# B&R Automation Studio project KeePakST401VersionX (part 4)

#### MbApp.st - Implementation code
```iecst
(********************************************************************
 * COPYRIGHT -- Bernecker + Rainer
 ********************************************************************
 * Program: MbApp
 * File: MbApp.st
 * Author: Bernecker + Rainer
 * Created: October 22, 2009
 ********************************************************************
 * Implementation of program MbApp
 * State Nomenclature: "request" is a write to the nordson melter asking for some data
 * 					   "read" is a read from the nordson melter of the previously requested data
 *                     "write" is a write to the nordson melter asking to write some data to the melter
 *                     "verify" is a read from the nordson melter where we check to see that the write was accepted
 ********************************************************************)

PROGRAM _INIT

	NordsonTxPacket.Byte0_MelterControl := 16#1;
	NordsonTxPacket.Byte1_Command := 3;
	NordsonTxPacket.Byte2_Data_Index := 16#78;
	NordsonTxPacket.Byte3_Channel_Num := 16#3;
	NordsonTxPacket.Byte4_5_WriteData := 0;
	NordsonTxPacket.Byte6_7_Mot1Spd := 0;
	NordsonTxPacket.Byte8_9_Mot2Spd := 0;
	NordsonTxPacket.Byte10_11_Mot3Spd := 0;
	NordsonTxPacket.Byte12_13_Mot4Spd := 0;
	NordsonTxPacket.Byte14_15_NotUsed := 0;

	state := MB_IDLE;

	(* init values *)
	mb_station 			:= 'IF2.ST2';					(* path to modbus station *)
	write_register_address	:= 1024;						(* register address on modbus station *)
	read_register_address	:= 0;						(* register address on modbus station *)
	num_registers_to_write := 8;
	num_registers_to_read := 8;

	testChannel := CHANNEL_ACT_TEMP_START;
	testIdx := IDX_ACT_TEMP;

	gAdhesiveCtrlInterface.Commands.MelterOn := TRUE;
	gAdhesiveCtrlInterface.Commands.PumpsOn := TRUE;
	gAdhesiveCtrlInterface.Parameters.NordsonComms.StandbyTimeoutTime := T#2h;

	FirstTimeCopySetTemps := FALSE;

END_PROGRAM

PROGRAM _CYCLIC

	IF(gAdhesiveCtrlInterface.Parameters.FeedbackIsModbusTCP) THEN
		gHMI.StatusDatapoints.NordsonModbusSDP := UNHIDE + UNLOCK;
	ELSE
		gHMI.StatusDatapoints.NordsonModbusSDP := HIDE + LOCK;
	END_IF

	StandbyTimer.IN := NOT(gRamCtrlInterface.Status.Running) AND NOT(gAdhesiveCtrlInterface.Commands.MelterStandbyOn);
	StandbyTimer.PT := gAdhesiveCtrlInterface.Parameters.NordsonComms.StandbyTimeoutTime;
	StandbyTimer();

	IF(StandbyTimer.Q) THEN
		gAdhesiveCtrlInterface.Commands.MelterStandbyOn := TRUE;
	END_IF

	//clearing standby on command shiuld turn standby off. Changed standbyoff to True
	IF(gAdhesiveCtrlInterface.Commands.MelterStandbyOff) THEN
		gAdhesiveCtrlInterface.Commands.MelterStandbyOff := TRUE;
		gAdhesiveCtrlInterface.Commands.MelterStandbyOn := FALSE;
	END_IF

	IF((gAdhesiveCtrlInterface.Status.NordsonInStandby) AND (gAdhesiveCtrlInterface.Parameters.FeedbackIsModbusTCP)) THEN
		gHMI.StatusDatapoints.NordsonStandbyOffSDP := UNHIDE + UNLOCK;
	ELSE
		gHMI.StatusDatapoints.NordsonStandbyOffSDP := HIDE + LOCK;
	END_IF

	//if nordson feedback is bypassed, the error count should reset to 0
	IF gAdhesiveCtrlInterface.Parameters.NordsonComms.ByPassFeedback THEN
		gAdhesiveCtrlInterface.Parameters.NordsonComms.ConsecutiveErrorCount := 0;
	END_IF

	CASE state OF

		MB_IDLE:
			FeedbackCycleTimer.IN := ((gAdhesiveCtrlInterface.Parameters.FeedbackIsModbusTCP) AND (gAdhesiveCtrlInterface.Parameters.NordsonComms.ByPassFeedback = FALSE));

			IF(gAdhesiveCtrlInterface.Parameters.FeedbackIsModbusTCP = FALSE) THEN
				gAdhesiveCtrlInterface.Parameters.NordsonComms.ConsecutiveErrorCount := 0;
			END_IF

			IF(gAdhesiveCtrlInterface.Commands.WriteChannelTemp) THEN
				gAdhesiveCtrlInterface.Commands.WriteChannelTemp := FALSE;
				TempChannelToWrite := 0;
				state := MB_WRITE_SET_TEMP;

			ELSIF(FeedbackCycleTimer.Q) THEN
				FeedbackCycleTimer.IN := FALSE;
				state := MB_REQUEST_MELTER_STATUS;
			END_IF

		MB_REQUEST_MELTER_STATUS:

			WriteMultipleRegisters.enable := 1;
			NordsonTxPacket.Byte0_MelterControl := MelterCmd;
			NordsonTxPacket.Byte1_Command := READ_COMMAND;
			NordsonTxPacket.Byte2_Data_Index := IDX_MELTER_STATUS;
			NordsonTxPacket.Byte3_Channel_Num := 0;

			IF((WriteMultipleRegisters.status = ERR_FUB_ENABLE_FALSE) OR (WriteMultipleRegisters.status = ERR_FUB_BUSY)) THEN
				//do nothing
			ELSIF(WriteMultipleRegisters.status = ERR_OK) THEN
				WriteMultipleRegisters.enable := 0;
				state := MB_READ_MELTER_STATUS;
			ELSE
				WriteMultipleRegisters.enable := 0;
				MBError := WriteMultipleRegisters.status;
				state := MB_ERROR;
			END_IF

		MB_READ_MELTER_STATUS:

			ReadMultipleRegisters.enable := 1;

			IF((ReadMultipleRegisters.status = ERR_FUB_ENABLE_FALSE) OR (ReadMultipleRegisters.status = ERR_FUB_BUSY)) THEN
				//do nothing
			ELSIF(ReadMultipleRegisters.status = ERR_OK) THEN

				ReadMultipleRegisters.enable := 0;

				IF(NordsonRxPacket.Byte2_Ack_Data_Index = NordsonTxPacket.Byte2_Data_Index) THEN

					gAdhesiveCtrlInterface.Parameters.NordsonComms.MelterStatus := NordsonRxPacket.Byte4_5_Read_Data_0;
					gAdhesiveCtrlInterface.Parameters.NordsonComms.MelterIsOn := (gAdhesiveCtrlInterface.Parameters.NordsonComms.MelterStatus <> 8); //melter status == 8 => melter is not on

					DecodeStatus;

					//the melter MUST see a 0 for its ON command before it sees a 1. Send a 0 if the unit is faulted OR we have previously told it to turn on. and it never came on
				//	IF((gAdhesiveCtrlInterface.Parameters.NordsonComms.UnitFaulted) OR ((gAdhesiveCtrlInterface.Parameters.NordsonComms.MelterIsOn = FALSE) AND (NordsonTxPacket.Byte0_MelterControl.0 = TRUE))) THEN
					IF((gAdhesiveCtrlInterface.Parameters.NordsonComms.MelterIsOn = FALSE) AND (NordsonTxPacket.Byte0_MelterControl.0 = TRUE)) THEN
						MelterCmd := MELTER_OFF + PUMPS_OFF; //melter off, pumps off
					ELSE

						MelterCmd := 0;
						IF(gAdhesiveCtrlInterface.Commands.MelterOn) THEN
							MelterCmd := MelterCmd + MELTER_ON;
						END_IF

						IF((gAdhesiveCtrlInterface.Commands.PumpsOn) AND (gAdhesiveCtrlInterface.Status.UnitReady)) THEN
							MelterCmd := MelterCmd + PUMPS_ON; //only turn the pump on if the melter is ready
						END_IF

						IF((gAdhesiveCtrlInterface.Commands.MelterStandbyOn = FALSE) OR ((gAdhesiveCtrlInterface.Status.NordsonInStandby = FALSE) AND NordsonTxPacket.Byte0_MelterControl.6 = TRUE)) THEN
							//do not standby on
						ELSIF (gAdhesiveCtrlInterface.Commands.MelterStandbyOn = TRUE) THEN
							MelterCmd := MelterCmd + STANDBY_ON; //only turn the pump on if the melter is ready
						END_IF
					END_IF

					state := MB_REQUEST_SET_TEMPS;
				ELSE
					//stay in this state and re-execute read
				END_IF

			ELSE
				ReadMultipleRegisters.enable := 0;
				MBError := ReadMultipleRegisters.status;
				state := MB_ERROR;
			END_IF

		MB_REQUEST_SET_TEMPS:

			WriteMultipleRegisters.enable := 1;
			NordsonTxPacket.Byte0_MelterControl := MelterCmd;
			NordsonTxPacket.Byte1_Command := READ_COMMAND;
			NordsonTxPacket.Byte2_Data_Index := IDX_SET_TEMP;
			NordsonTxPacket.Byte3_Channel_Num := CHANNEL_SET_TEMP_START;

			IF((WriteMultipleRegisters.status = ERR_FUB_ENABLE_FALSE) OR (WriteMultipleRegisters.status = ERR_FUB_BUSY)) THEN
				//do nothing
			ELSIF(WriteMultipleRegisters.status = ERR_OK) THEN
				WriteMultipleRegisters.enable := 0;
				gAdhesiveCtrlInterface.Parameters.NordsonComms.ConsecutiveErrorCount := 0;
				state := MB_READ_SET_TEMPS;
			ELSE
				WriteMultipleRegisters.enable := 0;
				MBError := WriteMultipleRegisters.status;
				state := MB_ERROR;
			END_IF

		MB_READ_SET_TEMPS:

			ReadMultipleRegisters.enable := 1;

			IF((ReadMultipleRegisters.status = ERR_FUB_ENABLE_FALSE) OR (ReadMultipleRegisters.status = ERR_FUB_BUSY)) THEN
				//do nothing
			ELSIF(ReadMultipleRegisters.status = ERR_OK) THEN
				ReadMultipleRegisters.enable := 0;
				gAdhesiveCtrlInterface.Parameters.NordsonComms.ConsecutiveErrorCount := 0;

				IF((NordsonRxPacket.Byte2_Ack_Data_Index = NordsonTxPacket.Byte2_Data_Index) AND
					(NordsonRxPacket.Byte3_Ack_Channel_Num = NordsonTxPacket.Byte3_Channel_Num)) THEN

					DecodeStatus;

					gAdhesiveCtrlInterface.Parameters.NordsonComms.ChannelSetTempActual[0] := NordsonRxPacket.Byte4_5_Read_Data_0;
					gAdhesiveCtrlInterface.Parameters.NordsonComms.ChannelSetTempActual[1] := NordsonRxPacket.Byte6_7_Read_Data_1;
					gAdhesiveCtrlInterface.Parameters.NordsonComms.ChannelSetTempActual[2] := NordsonRxPacket.Byte8_9_Read_Data_2;
					gAdhesiveCtrlInterface.Parameters.NordsonComms.ChannelSetTempActual[3] := NordsonRxPacket.Byte10_11_Read_Data_3;
					gAdhesiveCtrlInterface.Parameters.NordsonComms.ChannelSetTempActual[4] := NordsonRxPacket.Byte12_13_Read_Data_4;
					gAdhesiveCtrlInterface.Parameters.NordsonComms.ChannelSetTempActual[5] := NordsonRxPacket.Byte14_15_Read_Data_5;

					IF (FirstTimeCopySetTemps = FALSE) THEN
						gAdhesiveCtrlInterface.Parameters.NordsonComms.ChannelSetTempRequested := gAdhesiveCtrlInterface.Parameters.NordsonComms.ChannelSetTempActual;
						FirstTimeCopySetTemps := TRUE;
					END_IF

					state := MB_REQUEST_ACT_TEMPS; //for now, just go back to idle. Future versions need to read more stuff
				ELSE
					//stay in this state and re-execute read
				END_IF
			ELSE
				ReadMultipleRegisters.enable := 0;
				MBError := ReadMultipleRegisters.status;
				state := MB_ERROR;
			END_IF

		MB_REQUEST_ACT_TEMPS:

			WriteMultipleRegisters.enable := 1;
			NordsonTxPacket.Byte0_MelterControl := MelterCmd;
			NordsonTxPacket.Byte1_Command := READ_COMMAND;
			NordsonTxPacket.Byte2_Data_Index := IDX_ACT_TEMP;
			NordsonTxPacket.Byte3_Channel_Num := CHANNEL_ACT_TEMP_START;

			IF((WriteMultipleRegisters.status = ERR_FUB_ENABLE_FALSE) OR (WriteMultipleRegisters.status = ERR_FUB_BUSY)) THEN
				//do nothing
			ELSIF(WriteMultipleRegisters.status = ERR_OK) THEN
				WriteMultipleRegisters.enable := 0;
				state := MB_READ_ACT_TEMPS;
			ELSE
				WriteMultipleRegisters.enable := 0;
				MBError := WriteMultipleRegisters.status;
				state := MB_ERROR;
			END_IF

		MB_READ_ACT_TEMPS:

			ReadMultipleRegisters.enable := 1;

			IF((ReadMultipleRegisters.status = ERR_FUB_ENABLE_FALSE) OR (ReadMultipleRegisters.status = ERR_FUB_BUSY)) THEN
				//do nothing
			ELSIF(ReadMultipleRegisters.status = ERR_OK) THEN
				ReadMultipleRegisters.enable := 0;

				IF((NordsonRxPacket.Byte2_Ack_Data_Index = NordsonTxPacket.Byte2_Data_Index) AND
					(NordsonRxPacket.Byte3_Ack_Channel_Num = NordsonTxPacket.Byte3_Channel_Num)) THEN

					DecodeStatus;

					gAdhesiveCtrlInterface.Parameters.NordsonComms.ChannelActTemp[0] := NordsonRxPacket.Byte4_5_Read_Data_0;
					gAdhesiveCtrlInterface.Parameters.NordsonComms.ChannelActTemp[1] := NordsonRxPacket.Byte6_7_Read_Data_1;
					gAdhesiveCtrlInterface.Parameters.NordsonComms.ChannelActTemp[2] := NordsonRxPacket.Byte8_9_Read_Data_2;
					gAdhesiveCtrlInterface.Parameters.NordsonComms.ChannelActTemp[3] := NordsonRxPacket.Byte10_11_Read_Data_3;
					gAdhesiveCtrlInterface.Parameters.NordsonComms.ChannelActTemp[4] := NordsonRxPacket.Byte12_13_Read_Data_4;
					gAdhesiveCtrlInterface.Parameters.NordsonComms.ChannelActTemp[5] := NordsonRxPacket.Byte14_15_Read_Data_5;

					state := MB_REQUEST_ATS_ALARMS;
				ELSE
					//stay in this state and re-execute read
				END_IF

			ELSE
				ReadMultipleRegisters.enable := 0;
				MBError := ReadMultipleRegisters.status;
				state := MB_ERROR;
			END_IF

		MB_REQUEST_ATS_ALARMS:

			WriteMultipleRegisters.enable := 1;
			NordsonTxPacket.Byte0_MelterControl := MelterCmd;
			NordsonTxPacket.Byte1_Command := READ_COMMAND;
			NordsonTxPacket.Byte2_Data_Index := IDX_ATS_ALARMS;

			IF((WriteMultipleRegisters.status = ERR_FUB_ENABLE_FALSE) OR (WriteMultipleRegisters.status = ERR_FUB_BUSY)) THEN
				//do nothing
			ELSIF(WriteMultipleRegisters.status = ERR_OK) THEN
				WriteMultipleRegisters.enable := 0;
				state := MB_READ_ATS_ALARMS;
			ELSE
				WriteMultipleRegisters.enable := 0;
				MBError := WriteMultipleRegisters.status;
				state := MB_ERROR;
			END_IF

		MB_READ_ATS_ALARMS:

			ReadMultipleRegisters.enable := 1;

			IF((ReadMultipleRegisters.status = ERR_FUB_ENABLE_FALSE) OR (ReadMultipleRegisters.status = ERR_FUB_BUSY)) THEN
				//do nothing
			ELSIF(ReadMultipleRegisters.status = ERR_OK) THEN
				ReadMultipleRegisters.enable := 0;

				IF(NordsonRxPacket.Byte2_Ack_Data_Index = NordsonTxPacket.Byte2_Data_Index) THEN

					DecodeStatus;

					gAdhesiveCtrlInterface.Status.ATS_AddOnOverLimit := NordsonRxPacket.Byte4_5_Read_Data_0.0;
					gAdhesiveCtrlInterface.Status.ATS_AddOnUnderLimit := NordsonRxPacket.Byte4_5_Read_Data_0.1;

					state := MB_IDLE;
				ELSE
					//stay in this state and re-execute read
				END_IF

			ELSE
				ReadMultipleRegisters.enable := 0;
				MBError := ReadMultipleRegisters.status;
				state := MB_ERROR;
			END_IF

		MB_WRITE_SET_TEMP:

			WriteMultipleRegisters.enable := 1;
			NordsonTxPacket.Byte0_MelterControl := MelterCmd;
			NordsonTxPacket.Byte1_Command := WRITE_COMMAND;
			NordsonTxPacket.Byte2_Data_Index := IDX_SET_TEMP;
			NordsonTxPacket.Byte3_Channel_Num := TempChannelToWrite + 1; //TempChannelToWrite starts counting at 0, but nordson melter starts counting at 1
			NordsonTxPacket.Byte4_5_WriteData := gAdhesiveCtrlInterface.Parameters.NordsonComms.ChannelSetTempRequested[TempChannelToWrite];

			IF((WriteMultipleRegisters.status = ERR_FUB_ENABLE_FALSE) OR (WriteMultipleRegisters.status = ERR_FUB_BUSY)) THEN
				//do nothing
			ELSIF(WriteMultipleRegisters.status = ERR_OK) THEN
				WriteMultipleRegisters.enable := 0;
				state := MB_VERIFY_SET_TEMP_WRITE;
			ELSE
				WriteMultipleRegisters.enable := 0;
				MBError := WriteMultipleRegisters.status;
				state := MB_ERROR;
			END_IF

		MB_VERIFY_SET_TEMP_WRITE:

			ReadMultipleRegisters.enable := 1;

			IF((ReadMultipleRegisters.status = ERR_FUB_ENABLE_FALSE) OR (ReadMultipleRegisters.status = ERR_FUB_BUSY)) THEN
				//do nothing
			ELSIF(ReadMultipleRegisters.status = ERR_OK) THEN
				ReadMultipleRegisters.enable := 0;

				IF((NordsonRxPacket.Byte2_Ack_Data_Index = NordsonTxPacket.Byte2_Data_Index) AND
					(NordsonRxPacket.Byte3_Ack_Channel_Num = NordsonTxPacket.Byte3_Channel_Num)) THEN

					DecodeStatus;

					IF(TempChannelToWrite < NUM_NORDSON_TEMP_ZONES_M1) THEN
						IF(TempChannelToWrite = 0) THEN
							TempChannelToWrite := 2; //channel 0 and 1 get the same temp, no need to re-write channel 1
							state := MB_WRITE_SET_TEMP;
						ELSE
							TempChannelToWrite := TempChannelToWrite + 1; //set the temperature for the next channel (Skip channel 2). Machine has 3 total channels
							state := MB_WRITE_SET_TEMP;
						END_IF
					ELSE
						state := MB_IDLE;
					END_IF
				ELSE
					//stay in this state and re-execute read
				END_IF

			ELSE
				ReadMultipleRegisters.enable := 0;
				MBError := ReadMultipleRegisters.status;
				state := MB_ERROR;
			END_IF

		MB_REQUEST_ADH_USE:

			WriteMultipleRegisters.enable := 1;
			NordsonTxPacket.Byte0_MelterControl := MelterCmd;
			NordsonTxPacket.Byte1_Command := READ_COMMAND;
			NordsonTxPacket.Byte2_Data_Index := IDX_ADHESIVE_HOUR;
			NordsonTxPacket.Byte3_Channel_Num := CHANNEL_ADHESIVE_HOUR;

			IF((WriteMultipleRegisters.status = ERR_FUB_ENABLE_FALSE) OR (WriteMultipleRegisters.status = ERR_FUB_BUSY)) THEN
				//do nothing
			ELSIF(WriteMultipleRegisters.status = ERR_OK) THEN
				WriteMultipleRegisters.enable := 0;
				state := MB_READ_ACT_TEMPS;
			ELSE
				WriteMultipleRegisters.enable := 0;
				MBError := WriteMultipleRegisters.status;
				state := MB_ERROR;
			END_IF

		MB_READ_ADH_USE:

			ReadMultipleRegisters.enable := 1;

			IF((ReadMultipleRegisters.status = ERR_FUB_ENABLE_FALSE) OR (ReadMultipleRegisters.status = ERR_FUB_BUSY)) THEN
				//do nothing
			ELSIF(ReadMultipleRegisters.status = ERR_OK) THEN
				ReadMultipleRegisters.enable := 0;

				IF((NordsonRxPacket.Byte2_Ack_Data_Index = NordsonTxPacket.Byte2_Data_Index) AND
					(NordsonRxPacket.Byte3_Ack_Channel_Num = NordsonTxPacket.Byte3_Channel_Num)) THEN

					//	NordsonData.AdhesiveUsePerHour := NordsonRxPacket.Byte4_5_Read_Data_0 + (NordsonRxPacket.Byte6_7_Read_Data_1*(65536)); //data 0 + data 1 shifted up 16 bits

					state := MB_READ_ACT_TEMPS;
				ELSE
					//stay in this state and re-execute read
				END_IF
			END_IF

		MB_WRITE_REGISTERS:

			WriteMultipleRegisters.enable := 1;
			NordsonTxPacket.Byte0_MelterControl := MELTER_ON;
			NordsonTxPacket.Byte1_Command := READ_COMMAND;
			NordsonTxPacket.Byte2_Data_Index := testChannel;
			NordsonTxPacket.Byte3_Channel_Num := testIdx;

			IF((WriteMultipleRegisters.status = ERR_FUB_ENABLE_FALSE) OR (WriteMultipleRegisters.status = ERR_FUB_BUSY)) THEN
				//do nothing
			ELSIF(WriteMultipleRegisters.status = ERR_OK) THEN
				WriteMultipleRegisters.enable := 0;
				state := MB_READ_ACT_TEMPS;
			ELSE
				WriteMultipleRegisters.enable := 0;
				MBError := WriteMultipleRegisters.status;
				state := MB_ERROR;
			END_IF

		MB_READ_REGISTERS:

			ReadMultipleRegisters.enable := 1;

			IF((ReadMultipleRegisters.status = ERR_FUB_ENABLE_FALSE) OR (ReadMultipleRegisters.status = ERR_FUB_BUSY)) THEN
				//do nothing
			ELSIF(ReadMultipleRegisters.status = ERR_OK) THEN
				ReadMultipleRegisters.enable := 0;
				state := MB_IDLE;
			ELSE
				ReadMultipleRegisters.enable := 0;
				MBError := ReadMultipleRegisters.status;
				state := MB_ERROR;
			END_IF

		MB_ERROR:
			gAdhesiveCtrlInterface.Parameters.NordsonComms.ConsecutiveErrorCount := gAdhesiveCtrlInterface.Parameters.NordsonComms.ConsecutiveErrorCount + 1;
		state := MB_IDLE; //keep re-trying indefinetly, logic below will set/reset alarms alarm

	END_CASE;

	IF EDGEPOS(gAdhesiveCtrlInterface.Parameters.NordsonComms.ConsecutiveErrorCount >= 10) THEN
		MpAlarmXSet(gAlarmXCore, ALARM_NORDSON_COMMS);
	ELSIF EDGENEG(gAdhesiveCtrlInterface.Parameters.NordsonComms.ConsecutiveErrorCount >= 10)THEN
		MpAlarmXReset(gAlarmXCore, ALARM_NORDSON_COMMS);
	END_IF

	IF EDGEPOS(gAdhesiveCtrlInterface.Status.ATS_AddOnOverLimit) THEN
		MpAlarmXSet(gAlarmXCore, ALARM_ATS_OVERLIMIT);
	ELSIF EDGENEG(gAdhesiveCtrlInterface.Status.ATS_AddOnOverLimit)THEN
		MpAlarmXReset(gAlarmXCore, ALARM_ATS_OVERLIMIT);
	END_IF

	IF EDGEPOS(gAdhesiveCtrlInterface.Status.ATS_AddOnUnderLimit) THEN
		MpAlarmXSet(gAlarmXCore, ALARM_ATS_UNDERLIMIT);
	ELSIF EDGENEG(gAdhesiveCtrlInterface.Status.ATS_AddOnUnderLimit)THEN
		MpAlarmXReset(gAlarmXCore, ALARM_ATS_UNDERLIMIT);
	END_IF

	IF EDGEPOS(gAdhesiveCtrlInterface.Status.NordsonInStandby) THEN
		MpAlarmXSet(gAlarmXCore, ALARM_NORDSON_STANDBY);
	ELSIF EDGENEG(gAdhesiveCtrlInterface.Status.NordsonInStandby)THEN
		MpAlarmXReset(gAlarmXCore, ALARM_NORDSON_STANDBY);
	END_IF

	//force unit ready and unit faulted status flags if ModbusTCP control is selected and bypass is enabled
	IF(gAdhesiveCtrlInterface.Parameters.FeedbackIsModbusTCP AND gAdhesiveCtrlInterface.Parameters.NordsonComms.ByPassFeedback) THEN
		gAdhesiveCtrlInterface.Parameters.NordsonComms.UnitReady := TRUE;
		gAdhesiveCtrlInterface.Parameters.NordsonComms.UnitFaulted := FALSE;
		gAdhesiveCtrlInterface.Status.ATS_AddOnOverLimit := FALSE;
		gAdhesiveCtrlInterface.Status.ATS_AddOnUnderLimit := FALSE;
	END_IF

	//Must be called after state machine. Do not move any function calls that are already below this line
	WriteMultipleRegisters.pStation := ADR(mb_station);
	WriteMultipleRegisters.startAddress := write_register_address;
	WriteMultipleRegisters.nrRegisters := num_registers_to_write;
	WriteMultipleRegisters.pData := ADR(NordsonTxPacket);
	WriteMultipleRegisters.dataSize := SIZEOF(NordsonTxPacket);
	WriteMultipleRegisters();

	ReadMultipleRegisters.pStation := ADR(mb_station);
	ReadMultipleRegisters.startAddress := read_register_address;
	ReadMultipleRegisters.nrRegisters := num_registers_to_read;
	ReadMultipleRegisters.pData := ADR(NordsonRxPacket);
	ReadMultipleRegisters.dataSize := SIZEOF(NordsonRxPacket);
	ReadMultipleRegisters();

	FeedbackCycleTimer.PT := gAdhesiveCtrlInterface.Parameters.NordsonComms.FeedbackTime;
	FeedbackCycleTimer();

				END_PROGRAM
```

#### MbApp.typ - Local data types
```iecst
(********************************************************************
 * COPYRIGHT -- Bernecker + Rainer
 ********************************************************************
 * Program: MbApp
 * File: MbApp.typ
 * Author: Bernecker + Rainer
 * Created: October 22, 2009
 ********************************************************************
 * Local data types of program MbApp
 ********************************************************************)

TYPE
	ModbusTCP_Handling_States_enum :
		(
		MB_IDLE := 0,
		MB_REQUEST_SET_TEMPS,
		MB_READ_SET_TEMPS,
		MB_REQUEST_ACT_TEMPS,
		MB_READ_ACT_TEMPS,
		MB_REQUEST_MELTER_STATUS,
		MB_READ_MELTER_STATUS,
		MB_REQUEST_ADH_USE,
		MB_READ_ADH_USE,
		MB_WRITE_REGISTERS,
		MB_READ_REGISTERS,
		MB_REQUEST_MACHINE_STATUS,
		MB_WRITE_SET_TEMP,
		MB_VERIFY_SET_TEMP_WRITE,
		MB_REQUEST_ATS_ALARMS,
		MB_READ_ATS_ALARMS,
		MB_ERROR := 999
		);
END_TYPE
```

#### MbApp.var - Local variables
```iecst
(********************************************************************
 * COPYRIGHT -- Bernecker + Rainer
 ********************************************************************
 * Program: MbApp
 * File: MbApp.var
 * Author: Bernecker + Rainer
 * Created: October 22, 2009
 ********************************************************************
 * Local variables of program MbApp
 ********************************************************************)
VAR
	state : ModbusTCP_Handling_States_enum;
	mb_station : STRING[50];
	write_register_address : UINT;
	num_registers_to_write : UINT;
	read_register_address : UINT;
	num_registers_to_read : UINT;
	ReadMultipleRegisters : mbReadHoldingRegisters;
	WriteMultipleRegisters : mbWriteMultipleRegisters;
	MBError : UINT;
	testIdx : USINT;
	NordsonRxPacket : NordsonRxPacket_typ;
	testChannel : USINT;
	NordsonTxPacket : NordsonTxPacket_typ;
	FeedbackCycleTimer : TON;
	MelterCmd : USINT;
	TempChannelToWrite : USINT;
	StandbyTimer : TON;
	FirstTimeCopySetTemps : BOOL;
END_VAR
```

#### Action.st
```iecst
ACTION DecodeStatus:

	gAdhesiveCtrlInterface.Parameters.NordsonComms.UnitReady := NordsonRxPacket.Byte0_1_Status.0; //status word description from nordson manual
	gAdhesiveCtrlInterface.Parameters.NordsonComms.PumpStartUpProtectionOn := NordsonRxPacket.Byte0_1_Status.1;
	gAdhesiveCtrlInterface.Parameters.NordsonComms.Alert := NordsonRxPacket.Byte0_1_Status.2;
	gAdhesiveCtrlInterface.Parameters.NordsonComms.UnitFaulted := NordsonRxPacket.Byte0_1_Status.3;
	gAdhesiveCtrlInterface.Parameters.NordsonComms.ShutDown := NordsonRxPacket.Byte0_1_Status.4;
	gAdhesiveCtrlInterface.Parameters.NordsonComms.HeatUpPhaseActive := NordsonRxPacket.Byte0_1_Status.5;
	gAdhesiveCtrlInterface.Status.NordsonInStandby := NordsonRxPacket.Byte0_1_Status.6;
	gAdhesiveCtrlInterface.Parameters.NordsonComms.CommFault := NordsonRxPacket.Byte0_1_Status.14;
	gAdhesiveCtrlInterface.Parameters.NordsonComms.CommFaultInDataValue := NordsonRxPacket.Byte0_1_Status.15;

END_ACTION
```

### Program Logical/Actuators/NordsonComm/NordsonExtendedComm (IEC)

#### MbPressure.st - Init, cyclic, exit code
```iecst
(*********************************************************************************
 * Copyright: B&R Industrial Automation GmbH
 * Author:    nealj
 * Created:   May 27, 2021/1:33 PM
 * This task will cyclicly read the current pressure and the tank level and will
 * write the pressure setpoints.
 *********************************************************************************)

PROGRAM _INIT

    Station              := 'IF2.ST2';
    ModbusRead.pStation  := ADR(Station);
    ModbusWrite.pStation := ADR(Station);

END_PROGRAM

PROGRAM _CYCLIC

    Channel.PressureSetpoint := PressureSetpoint;

    CASE ExtendedCommsState OF

        WORD_MANIPULATION:
            Channel.ActualPressure           := (UDINT_TO_REAL(Registers.ChannelActualPressureWord) / 1000);
            Tank.ActualLevel                    := Registers.TankActualLevelWord;
            Registers.ChannelSetPressureWord := REAL_TO_UDINT(Channel.PressureSetpoint * 1000);
            ExtendedCommsState                  := READ_ACTPRESS_W1;

        READ_ACTPRESS_W1:
            IF (ModbusRead.status = ERR_OK) THEN
                ModbusRead.enable  := FALSE;
                ExtendedCommsState := WRITE_SETPRESS_W1;
            ELSIF (ModbusRead.status = ERR_FUB_ENABLE_FALSE) THEN
                ModbusRead.startAddress := 6103;
                ModbusRead.nrRegisters  := 2;
                ModbusRead.pData        := ADR(Registers.ChannelActualPressureWord);
                ModbusRead.dataSize     := 8;
                ModbusRead.enable       := TRUE;
            END_IF

        WRITE_SETPRESS_W1:
            IF (ModbusWrite.status = ERR_OK) THEN
                ModbusWrite.enable  := FALSE;
                ExtendedCommsState := READ_TANKLEVEL_W1;
            ELSIF (ModbusRead.status = ERR_FUB_ENABLE_FALSE) AND (WriteFlag) THEN
                ModbusWrite.startAddress := 6203;
                ModbusWrite.nrRegisters  := 2;
                ModbusWrite.pData        := ADR(Registers.ChannelSetPressureWord);
                ModbusWrite.dataSize     := 8;
                ModbusWrite.enable       := TRUE;
                WriteFlag              := FALSE;
            ELSIF (ModbusWrite.status = ERR_FUB_ENABLE_FALSE) AND NOT(WriteFlag) THEN
                ExtendedCommsState := READ_TANKLEVEL_W1;
            END_IF

        READ_TANKLEVEL_W1:
            IF (ModbusRead.status = ERR_OK) THEN
                ModbusRead.enable := FALSE;
                ExtendedCommsState := WORD_MANIPULATION;
            ELSIF (ModbusWrite.status = ERR_FUB_ENABLE_FALSE) THEN
                ModbusRead.startAddress := 13002;
                ModbusRead.nrRegisters  := 1;
                ModbusRead.pData        := ADR(Registers.TankActualLevelWord);
                ModbusRead.dataSize     := 4;
                ModbusRead.enable       := TRUE;
            END_IF

        MODBUS_ERROR:
            IF ((ModbusRead.status = ERR_FUB_ENABLE_FALSE) AND (ModbusWrite.status = ERR_FUB_ENABLE_FALSE)) THEN
                ExtendedCommsState := WORD_MANIPULATION;
            ELSE
                ReadErrorNumber    := ModbusRead.status;
                WriteErrorNumber   := ModbusWrite.status;
                ModbusRead.enable  := FALSE;
                ModbusWrite.enable := FALSE;
            END_IF

    END_CASE

    IF ((ModbusRead.status > 0) AND (ModbusRead.status < 65534)) OR ((ModbusWrite.status > 0) AND (ModbusWrite.status < 65534)) THEN
        ExtendedCommsState := MODBUS_ERROR;
    END_IF

    //Call FUBs
    ModbusRead();
    ModbusWrite();

END_PROGRAM

PROGRAM _EXIT

END_PROGRAM
```

#### Types.typ - Local data types
```iecst
TYPE
	ExtendedComms_enum :
		(
		WORD_MANIPULATION,
		READ_ACTPRESS_W1,
		READ_ACTPRESS_W2,
		READ_ACTPRESS_W3,
		READ_ACTPRESS_W4,
		WRITE_SETPRESS_W1,
		WRITE_SETPRESS_W2,
		WRITE_SETPRESS_W3,
		WRITE_SETPRESS_W4,
		READ_TANKLEVEL_W1,
		MODBUS_ERROR
		);
END_TYPE
```

#### Variables.var - Local variables
```iecst
VAR
	ModbusRead : mbReadHoldingRegisters;
	ModbusWrite : mbWriteMultipleRegisters;
	Station : STRING[10];
	Registers : Register_typ;
	Channel : Channel_typ;
	PressureSetpoint : REAL;
	Tank : Tank_typ;
	ExtendedCommsState : ExtendedComms_enum;
	WriteFlag : BOOL;
	ReadErrorNumber : UINT;
	WriteErrorNumber : UINT;
	New_Variable : USINT;
END_VAR
```

### Program Logical/Actuators/FlexTest (IEC)

#### Variables.var
```iecst
VAR
	FB_NDSN_MB_PBFlex_Proc : FB_NDSN_MB_PBFlex_Process;
	FB_NDSN_MB_PBFlex_Ctrl : FB_NDSN_MB_PBFlex_CtrlSts;
	mb_Station : STRING[30];
END_VAR
```

#### Main.st
```iecst
PROGRAM _INIT
	(* Insert code here *)
	b_ModuleStatus;
	mb_Station 			:= 'IF2.ST2';
    Melter;
 //   FB_NDSN_MB_PBFlex_Ctrl;
 //   FB_NDSN_MB_PBFlex_Proc;
END_PROGRAM

PROGRAM _CYCLIC
	(* Insert code here *)
//	FB_NDSN_MB_PBFlex_Ctrl(IN_b_Enable :=NOT  Melter.b_r_LostCommunication,	IN_mb_station := mb_Station,Melter := Melter);
//  FB_NDSN_MB_PBFlex_Proc(IN_b_Enable :=NOT  Melter.b_r_LostCommunication, IN_mb_station := mb_Station,Melter := Melter);
//  Melter.b_r_LostCommunication :=NOT b_ModuleStatus;

    FB_NDSN_MB_PBFlex_Ctrl(IN_b_Enable := NOT Melter.b_r_LostCommunication , IN_mb_station := mb_Station , Melter := Melter );
    FB_NDSN_MB_PBFlex_Proc(IN_b_Enable := NOT Melter.b_r_LostCommunication , IN_mb_station := mb_Station , Melter := Melter );
    Melter.b_r_LostCommunication := NOT b_ModuleStatus;

END_PROGRAM

PROGRAM _EXIT
	(* Insert code here *)

END_PROGRAM
```

### Program Logical/Recipes/Recipes (IEC)

#### Variables.var
```iecst
VAR
	LastRecipeLoaded : STRING[80];
	MpRecipeXml_0 : MpRecipeXml;
	MpRecipeRegPar_0 : MpRecipeRegPar;
	MpRecipeRegPar_1 : MpRecipeRegPar;
	MpRecipeRegPar_2 : MpRecipeRegPar;
	MpRecipeRegPar_3 : MpRecipeRegPar;
	MpRecipeRegPar_4 : MpRecipeRegPar;
	MpRecipeRegPar_5 : MpRecipeRegPar;
	RegParActive0 : BOOL;
	RegParActive1 : BOOL;
	RegParActive2 : BOOL;
	RegParActive3 : BOOL;
	RegParActive4 : BOOL;
	RegParActive5 : BOOL;
	AllParsRegistered : BOOL;
END_VAR
```

#### Cyclic.ld
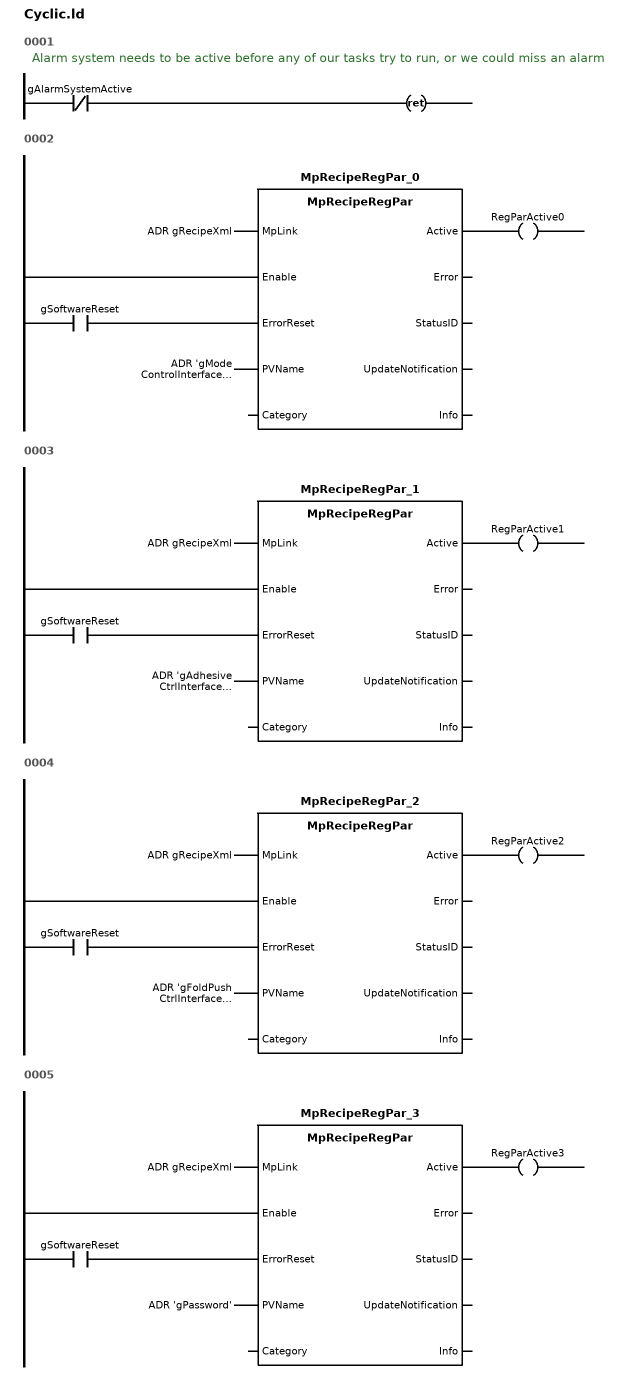
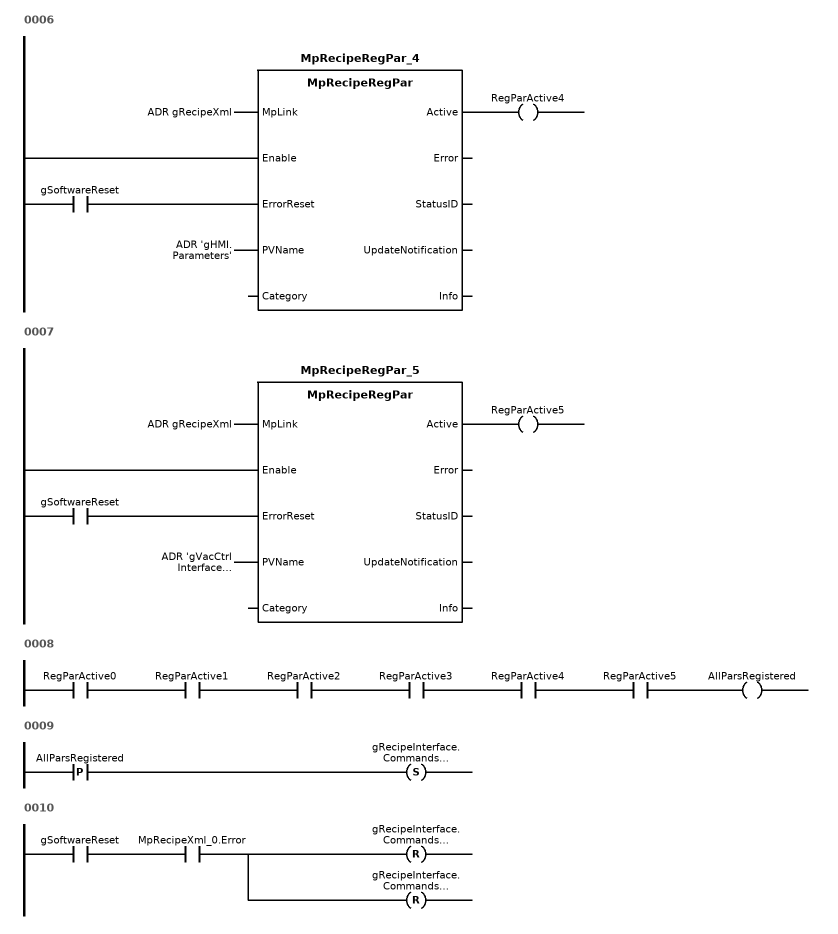
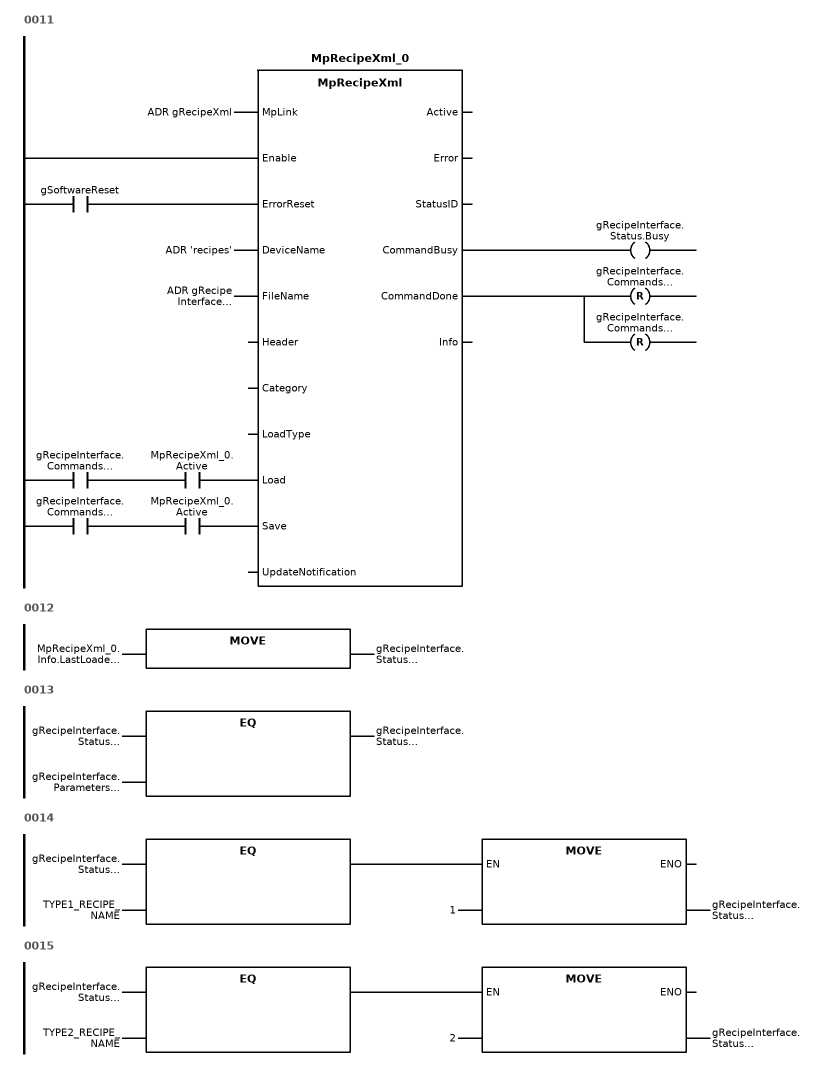
Ladder, written as Structured Text:
```iecst
PROGRAM _CYCLIC
VAR
    _e1 : R_TRIG;
    _p2 : BOOL;
    _p3 : BOOL;
END_VAR
(* Network 1: Alarm system needs to be active before any of our tasks try to run, or we could miss an alarm *)
IF NOT gAlarmSystemActive THEN RETURN; END_IF;

(* Network 2 *)
MpRecipeRegPar_0(MpLink := ADR(gRecipeXml), Enable := TRUE, ErrorReset := gSoftwareReset, PVName := ADR('gModeControlInterface.Parameters'));
RegParActive0 := MpRecipeRegPar_0.Active;

(* Network 3 *)
MpRecipeRegPar_1(MpLink := ADR(gRecipeXml), Enable := TRUE, ErrorReset := gSoftwareReset, PVName := ADR('gAdhesiveCtrlInterface.Parameters'));
RegParActive1 := MpRecipeRegPar_1.Active;

(* Network 4 *)
MpRecipeRegPar_2(MpLink := ADR(gRecipeXml), Enable := TRUE, ErrorReset := gSoftwareReset, PVName := ADR('gFoldPushCtrlInterface.Parameters'));
RegParActive2 := MpRecipeRegPar_2.Active;

(* Network 5 *)
MpRecipeRegPar_3(MpLink := ADR(gRecipeXml), Enable := TRUE, ErrorReset := gSoftwareReset, PVName := ADR('gPassword'));
RegParActive3 := MpRecipeRegPar_3.Active;

(* Network 6 *)
MpRecipeRegPar_4(MpLink := ADR(gRecipeXml), Enable := TRUE, ErrorReset := gSoftwareReset, PVName := ADR('gHMI.Parameters'));
RegParActive4 := MpRecipeRegPar_4.Active;

(* Network 7 *)
MpRecipeRegPar_5(MpLink := ADR(gRecipeXml), Enable := TRUE, ErrorReset := gSoftwareReset, PVName := ADR('gVacCtrlInterface.Parameters'));
RegParActive5 := MpRecipeRegPar_5.Active;

(* Network 8 *)
AllParsRegistered := RegParActive0 AND RegParActive1 AND RegParActive2 AND RegParActive3 AND RegParActive4 AND RegParActive5;

(* Network 9 *)
_e1(CLK := AllParsRegistered);
IF _e1.Q THEN gRecipeInterface.Commands.LoadRecipe := TRUE; END_IF;

(* Network 10 *)
IF gSoftwareReset AND MpRecipeXml_0.Error THEN
    gRecipeInterface.Commands.LoadRecipe := FALSE;
    gRecipeInterface.Commands.SaveRecipe := FALSE;
END_IF;

(* Network 11 *)
MpRecipeXml_0(MpLink := ADR(gRecipeXml), Enable := TRUE, ErrorReset := gSoftwareReset, DeviceName := ADR('recipes'), FileName := ADR(gRecipeInterface.Parameters.RecipeName), Load := gRecipeInterface.Commands.LoadRecipe AND MpRecipeXml_0.Active, Save := gRecipeInterface.Commands.SaveRecipe AND MpRecipeXml_0.Active);
gRecipeInterface.Status.Busy := MpRecipeXml_0.CommandBusy;
IF MpRecipeXml_0.CommandDone THEN
    gRecipeInterface.Commands.LoadRecipe := FALSE;
    gRecipeInterface.Commands.SaveRecipe := FALSE;
END_IF;

(* Network 12 *)
gRecipeInterface.Status.LoadedRecipeName := MpRecipeXml_0.Info.LastLoadedRecipe;

(* Network 13 *)
gRecipeInterface.Status.RecipeHasBeenLoaded := gRecipeInterface.Status.LoadedRecipeName = gRecipeInterface.Parameters.RecipeName;

(* Network 14 *)
_p2 := gRecipeInterface.Status.LoadedRecipeName = TYPE1_RECIPE_NAME;
IF _p2 THEN gRecipeInterface.Status.LoadedRecipeIndex := 1; END_IF;

(* Network 15 *)
_p3 := gRecipeInterface.Status.LoadedRecipeName = TYPE2_RECIPE_NAME;
IF _p3 THEN gRecipeInterface.Status.LoadedRecipeIndex := 2; END_IF;
END_PROGRAM
```

#### Init.st
```iecst
PROGRAM _INIT
	(* Insert code here *)

	gRecipeInterface.Commands.LoadRecipe := 1; //load settings on startup

	IF gRecipeInterface.Parameters.RecipeName = '' THEN
		gRecipeInterface.Parameters.RecipeName := TYPE1_RECIPE_NAME;
	END_IF

	//If the last recipe was type 2, set file name to that recipe. Otherwise default to recipe 1 file name
//	IF LastRecipeLoaded = TYPE2_RECIPE_NAME THEN
//		gRecipeInterface.Parameters.RecipeName := TYPE2_RECIPE_NAME;
//	ELSE
//		gRecipeInterface.Parameters.RecipeName := TYPE1_RECIPE_NAME;
//	END_IF

END_PROGRAM
```

### Program Logical/Recipes/GluePattCtrl (IEC)

#### Cyclic.st - Cyclic code
```iecst
PROGRAM _CYCLIC

	SaveButton_RTrig.CLK := gRecipeInterface.Commands.SaveRecipe;

	IF SaveButton_RTrig.Q THEN
		gAdhesiveCtrlInterface.Parameters.SavedPatterns[gAdhesiveCtrlInterface.Parameters.PatternSelection].AdhesivePatterns := gAdhesiveCtrlInterface.Parameters.AdhesivePatterns;
	END_IF

	IF gHMI.StatusDatapoints.AdhesivePatternConfirmedSDP.0 THEN
		gAdhesiveCtrlInterface.Parameters.AdhesivePatterns := gAdhesiveCtrlInterface.Parameters.SavedPatterns[gAdhesiveCtrlInterface.Parameters.PatternSelection].AdhesivePatterns;
		gHMI.StatusDatapoints.AdhesivePatternConfirmedSDP.0 := FALSE;
	END_IF

    SaveButton_RTrig();

END_PROGRAM
```

#### Variables.var - Local variables
```iecst
VAR
	SaveButton_RTrig : R_TRIG;
END_VAR
```

### Program Logical/AlarmControl/AlarmHandling (IEC)

#### Cyclic.ld - Cyclic code
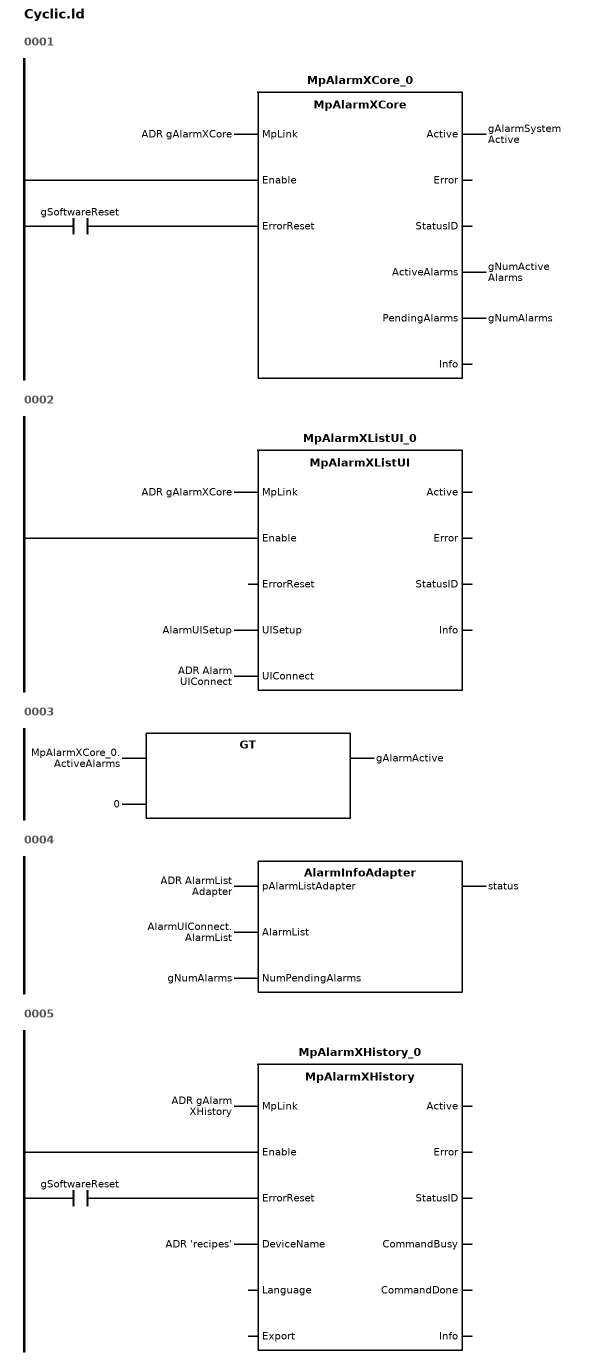
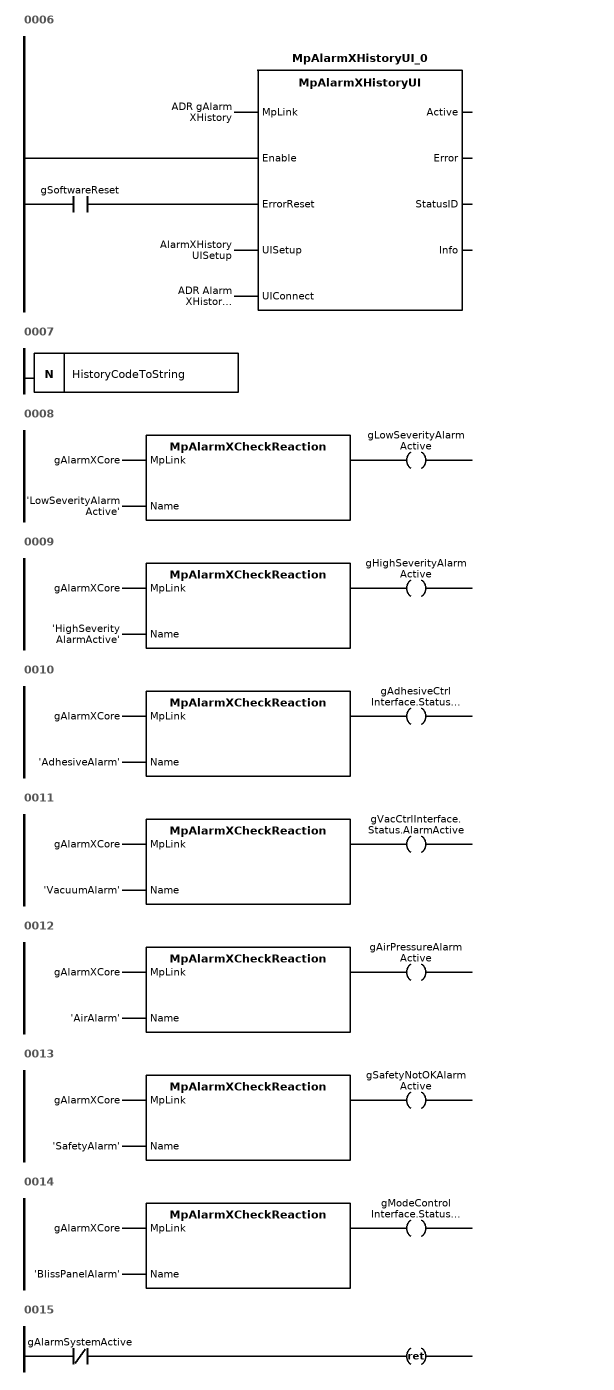
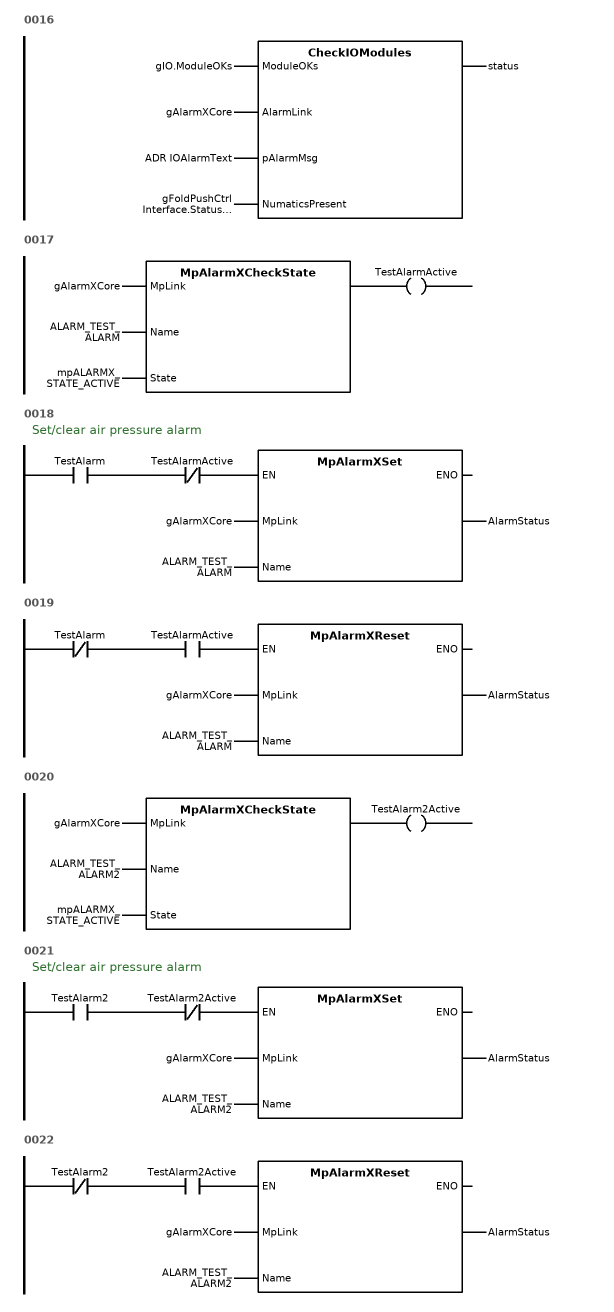
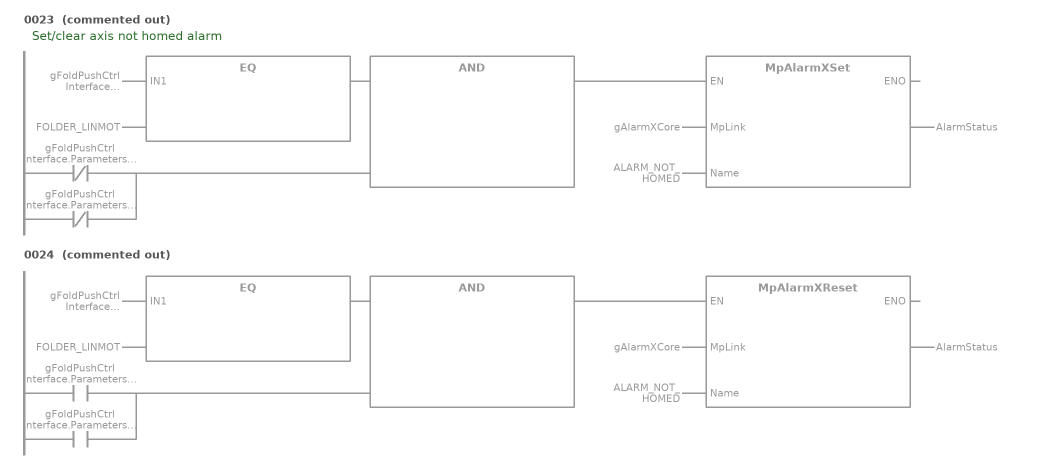
Ladder, written as Structured Text:
```iecst
PROGRAM _CYCLIC
(* Network 1 *)
MpAlarmXCore_0(MpLink := ADR(gAlarmXCore), Enable := TRUE, ErrorReset := gSoftwareReset);
gAlarmSystemActive := MpAlarmXCore_0.Active;
gNumActiveAlarms := MpAlarmXCore_0.ActiveAlarms;
gNumAlarms := MpAlarmXCore_0.PendingAlarms;

(* Network 2 *)
MpAlarmXListUI_0(MpLink := ADR(gAlarmXCore), Enable := TRUE, UISetup := AlarmUISetup, UIConnect := ADR(AlarmUIConnect));

(* Network 3 *)
gAlarmActive := MpAlarmXCore_0.ActiveAlarms > 0;

(* Network 4 *)
status := AlarmInfoAdapter(pAlarmListAdapter := ADR(AlarmListAdapter), AlarmList := AlarmUIConnect.AlarmList, NumPendingAlarms := gNumAlarms);

(* Network 5 *)
MpAlarmXHistory_0(MpLink := ADR(gAlarmXHistory), Enable := TRUE, ErrorReset := gSoftwareReset, DeviceName := ADR('recipes'));

(* Network 6 *)
MpAlarmXHistoryUI_0(MpLink := ADR(gAlarmXHistory), Enable := TRUE, ErrorReset := gSoftwareReset, UISetup := AlarmXHistoryUISetup, UIConnect := ADR(AlarmXHistoryUIConnect));

(* Network 7 *)
HistoryCodeToString;

(* Network 8 *)
gLowSeverityAlarmActive := MpAlarmXCheckReaction(MpLink := gAlarmXCore, Name := 'LowSeverityAlarmActive');

(* Network 9 *)
gHighSeverityAlarmActive := MpAlarmXCheckReaction(MpLink := gAlarmXCore, Name := 'HighSeverityAlarmActive');

(* Network 10 *)
gAdhesiveCtrlInterface.Status.AlarmActive := MpAlarmXCheckReaction(MpLink := gAlarmXCore, Name := 'AdhesiveAlarm');

(* Network 11 *)
gVacCtrlInterface.Status.AlarmActive := MpAlarmXCheckReaction(MpLink := gAlarmXCore, Name := 'VacuumAlarm');

(* Network 12 *)
gAirPressureAlarmActive := MpAlarmXCheckReaction(MpLink := gAlarmXCore, Name := 'AirAlarm');

(* Network 13 *)
gSafetyNotOKAlarmActive := MpAlarmXCheckReaction(MpLink := gAlarmXCore, Name := 'SafetyAlarm');

(* Network 14 *)
gModeControlInterface.Status.BlissPanelAlarmActive := MpAlarmXCheckReaction(MpLink := gAlarmXCore, Name := 'BlissPanelAlarm');

(* Network 15 *)
IF NOT gAlarmSystemActive THEN RETURN; END_IF;

(* Network 16 *)
status := CheckIOModules(ModuleOKs := gIO.ModuleOKs, AlarmLink := gAlarmXCore, pAlarmMsg := ADR(IOAlarmText), NumaticsPresent := gFoldPushCtrlInterface.Status.PowelinkConfig);

(* Network 17 *)
TestAlarmActive := MpAlarmXCheckState(MpLink := gAlarmXCore, Name := ALARM_TEST_ALARM, State := mpALARMX_STATE_ACTIVE);

(* Network 18: Set/clear air pressure alarm *)
IF TestAlarm AND NOT TestAlarmActive THEN
    AlarmStatus := MpAlarmXSet(MpLink := gAlarmXCore, Name := ALARM_TEST_ALARM);
END_IF;

(* Network 19 *)
IF NOT TestAlarm AND TestAlarmActive THEN
    AlarmStatus := MpAlarmXReset(MpLink := gAlarmXCore, Name := ALARM_TEST_ALARM);
END_IF;

(* Network 20 *)
TestAlarm2Active := MpAlarmXCheckState(MpLink := gAlarmXCore, Name := ALARM_TEST_ALARM2, State := mpALARMX_STATE_ACTIVE);

(* Network 21: Set/clear air pressure alarm *)
IF TestAlarm2 AND NOT TestAlarm2Active THEN
    AlarmStatus := MpAlarmXSet(MpLink := gAlarmXCore, Name := ALARM_TEST_ALARM2);
END_IF;

(* Network 22 *)
IF NOT TestAlarm2 AND TestAlarm2Active THEN
    AlarmStatus := MpAlarmXReset(MpLink := gAlarmXCore, Name := ALARM_TEST_ALARM2);
END_IF;

(* Network 23: Set/clear axis not homed alarm *) (* commented out *)
// IF (gFoldPushCtrlInterface.Parameters.FolderTypeSelection = FOLDER_LINMOT) AND (NOT gFoldPushCtrlInterface.Parameters.LinMotTopFolder.Status.IsHomed OR NOT gFoldPushCtrlInterface.Parameters.LinMotBotFolder.Status.IsHomed) THEN
//     AlarmStatus := MpAlarmXSet(MpLink := gAlarmXCore, Name := ALARM_NOT_HOMED);
// END_IF;

(* Network 24 *) (* commented out *)
// IF (gFoldPushCtrlInterface.Parameters.FolderTypeSelection = FOLDER_LINMOT) AND (gFoldPushCtrlInterface.Parameters.LinMotTopFolder.Status.IsHomed OR gFoldPushCtrlInterface.Parameters.LinMotBotFolder.Status.IsHomed) THEN
//     AlarmStatus := MpAlarmXReset(MpLink := gAlarmXCore, Name := ALARM_NOT_HOMED);
// END_IF;
END_PROGRAM
```

#### Init.st
```iecst
PROGRAM _INIT

	FOR i := 0 TO 99 DO
		gIO.ModuleOKs[i] := TRUE;
	END_FOR;

	IOAlarmText;

	AlarmXHistoryUISetup.AlarmListScrollWindow := 1;
	AlarmXHistoryUISetup.AlarmListSize := 6;

END_PROGRAM
```

#### Variables.var - Local variables
```iecst
VAR
	IOAlarmText : STRING[100];
	MpAlarmXCore_0 : MpAlarmXCore;
	MpAlarmXListUI_0 : MpAlarmXListUI;
	AlarmUISetup : MpAlarmXListUISetupType;
	AlarmUIConnect : MpAlarmXListUIConnectType;
	AlarmListAdapter : AlarmListAdapter_typ;
	AlarmHistoryListAdapter : AlarmListAdapter_typ;
	status : BOOL;
	i : UINT;
	MpAlarmXHistory_0 : MpAlarmXHistory;
	MpAlarmXHistoryUI_0 : MpAlarmXHistoryUI;
	AlarmXHistoryUIConnect : MpAlarmXHistoryUIConnectType;
	AlarmXHistoryUISetup : MpAlarmXHistoryUISetupType;
	AlarmStatus : DINT;
	TestAlarm2 : BOOL;
	TestAlarm : BOOL;
	TestAlarm2Active : BOOL;
	TestAlarmActive : BOOL;
END_VAR
```

#### LocalFunctions.fun
```iecst
FUNCTION AlarmInfoAdapter : BOOL (*Convert some alarm elements from Bool to Str*) (*$GROUP=User,$CAT=User,$GROUPICON=User.png,$CATICON=User.png*)
	VAR_INPUT
		pAlarmListAdapter : REFERENCE TO AlarmListAdapter_typ;
		AlarmList : MpAlarmXListUIAlarmListType;
		NumPendingAlarms : UDINT;
	END_VAR
	VAR
		i : UINT;
	END_VAR
END_FUNCTION

FUNCTION CheckIOModules : BOOL (*TODO: Add your comment here*) (*$GROUP=User,$CAT=User,$GROUPICON=User.png,$CATICON=User.png*)
	VAR_INPUT
		ModuleOKs : ARRAY[0..99] OF BOOL;
		AlarmLink : MpComIdentType;
		pAlarmMsg : UDINT;
	END_VAR
	VAR
		i : USINT;
	END_VAR
	VAR_INPUT
		NumaticsPresent : BOOL;
	END_VAR
END_FUNCTION
```

#### AlarmInfoAdapter.st
```iecst
(* Convert some alarm elements from Bool to Str *)
FUNCTION AlarmInfoAdapter

	IF(NumPendingAlarms = 0) THEN
		FOR i:= 0  TO 49 DO
			pAlarmListAdapter.Acknowledged[i] := '';
			pAlarmListAdapter.Active[i] := '';
			pAlarmListAdapter.Code[i] := '';
		END_FOR
	ELSE

		FOR i:=0 TO AlarmList.MaxSelection DO

			IF(AlarmList.StateAcknowledged[i] = TRUE) THEN
				pAlarmListAdapter.Acknowledged[i] := 'Yes';
			ELSE
				pAlarmListAdapter.Acknowledged[i] := 'No';
			END_IF

			IF(AlarmList.StateActive[i] = TRUE) THEN
				pAlarmListAdapter.Active[i] := 'Yes';
			ELSE
				pAlarmListAdapter.Active[i] := 'No';
			END_IF

			brsitoa(AlarmList.Code[i],ADR(pAlarmListAdapter.Code[i]));

		END_FOR;

		FOR i:= AlarmList.MaxSelection + 1  TO 49 DO
			pAlarmListAdapter.Acknowledged[i] := '';
			pAlarmListAdapter.Active[i] := '';
			pAlarmListAdapter.Code[i] := '';
		END_FOR

	END_IF

	AlarmInfoAdapter := TRUE;

END_FUNCTION
```

#### CheckIOModules.st
```iecst
(* TODO: Add your comment here *)
FUNCTION CheckIOModules

	brsmemset(pAlarmMsg, 0, 100);

	FOR i := 1 TO 99 DO

		IF(ModuleOKs[i] = FALSE) THEN

			IF (i = 1) THEN
				brsstrcat(pAlarmMsg, ADR ('Module 1 Bus Receiver'));
			ELSIF (i = 2) THEN
				brsstrcat(pAlarmMsg, ADR ('Module 2 DI 1'));
			ELSIF (i = 3) THEN
				brsstrcat(pAlarmMsg, ADR ('Module 3 D0 1'));
			ELSIF (i = 4) THEN
				brsstrcat(pAlarmMsg, ADR ('Module 4 DO 2(high wattage outputs)'));
			ELSIF (i = 5) THEN
				brsstrcat(pAlarmMsg, ADR ('Module 5 Encoder Inputs'));
			ELSIF (i = 6) THEN
				brsstrcat(pAlarmMsg, ADR ('SLX Module'));

			ELSIF (i = 7) THEN
				IF NumaticsPresent THEN
				brsstrcat(pAlarmMsg, ADR ('Module 7 Pneumatics 580'));
				END_IF

			END_IF

			IF (i=7 AND NumaticsPresent) OR (i<> 7) THEN
			brsstrcat(pAlarmMsg, ADR (' Not OK'));

			MpAlarmXSet(AlarmLink, ALARM_IO_MODULE_NOT_OK);
			END_IF

			RETURN;

		END_IF

	END_FOR;

	MpAlarmXReset(AlarmLink, ALARM_IO_MODULE_NOT_OK);

	CheckIOModules := 1;

END_FUNCTION
```

#### Action.st
```iecst
//convert alarm code integer into a string. This let's us completely clear alarm codes for empty entries instead of entering a '0'
ACTION HistoryCodeToString:

	FOR i:=0 TO AlarmXHistoryUIConnect.AlarmList.MaxSelection DO

		brsitoa(AlarmXHistoryUIConnect.AlarmList.Code[i], ADR(AlarmHistoryListAdapter.Code[i]));

	END_FOR;

	FOR i:= AlarmXHistoryUIConnect.AlarmList.MaxSelection + 1  TO 49 DO
		AlarmHistoryListAdapter.Code[i] := '';
	END_FOR

END_ACTION
```

### Program Logical/HMI/HMIControl (IEC)

#### Variables.var
```iecst
VAR
	FlashOFF : TON;
	FlashON : TON;
	status : BOOL;
	SettingsLoaded : BOOL;
	LogoutTimer : TON;
	OldPage : USINT;
	ResetTimeoutTimer : BOOL;
	ResetUserLevel : BOOL;
END_VAR
```

#### Cyclic.ld
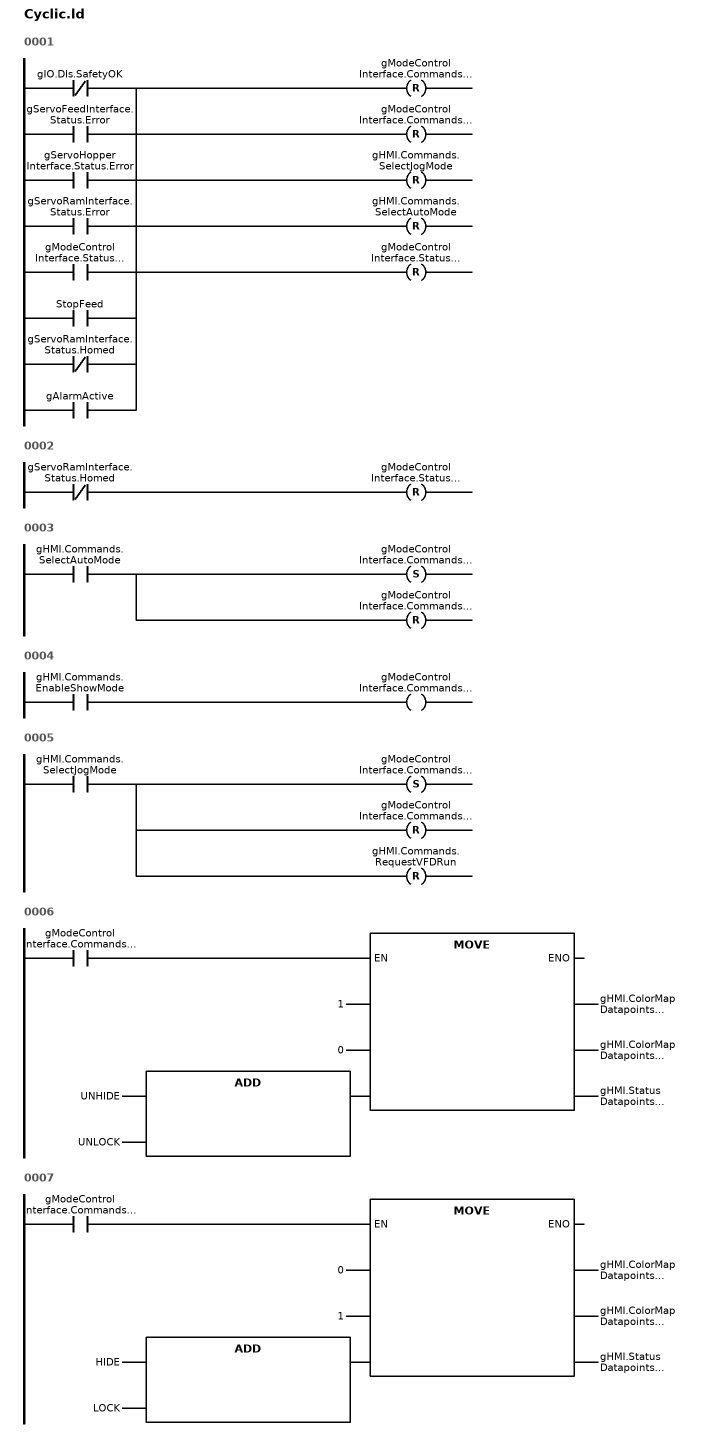
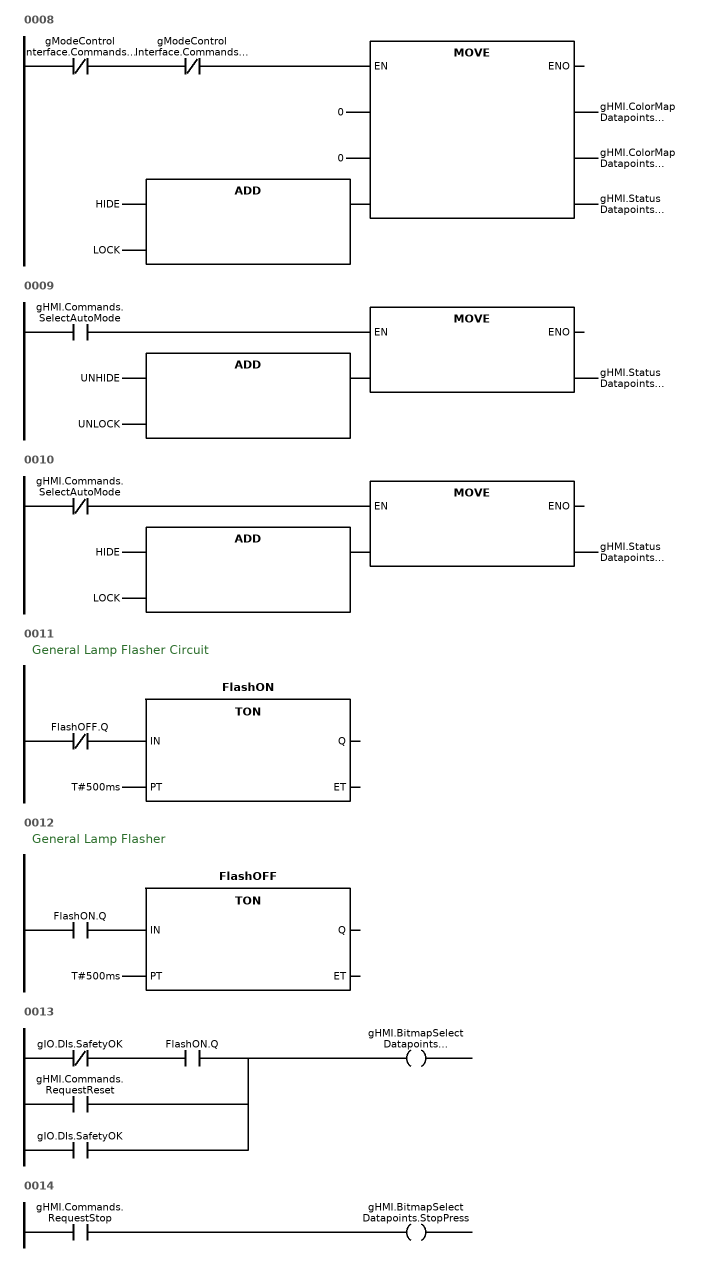
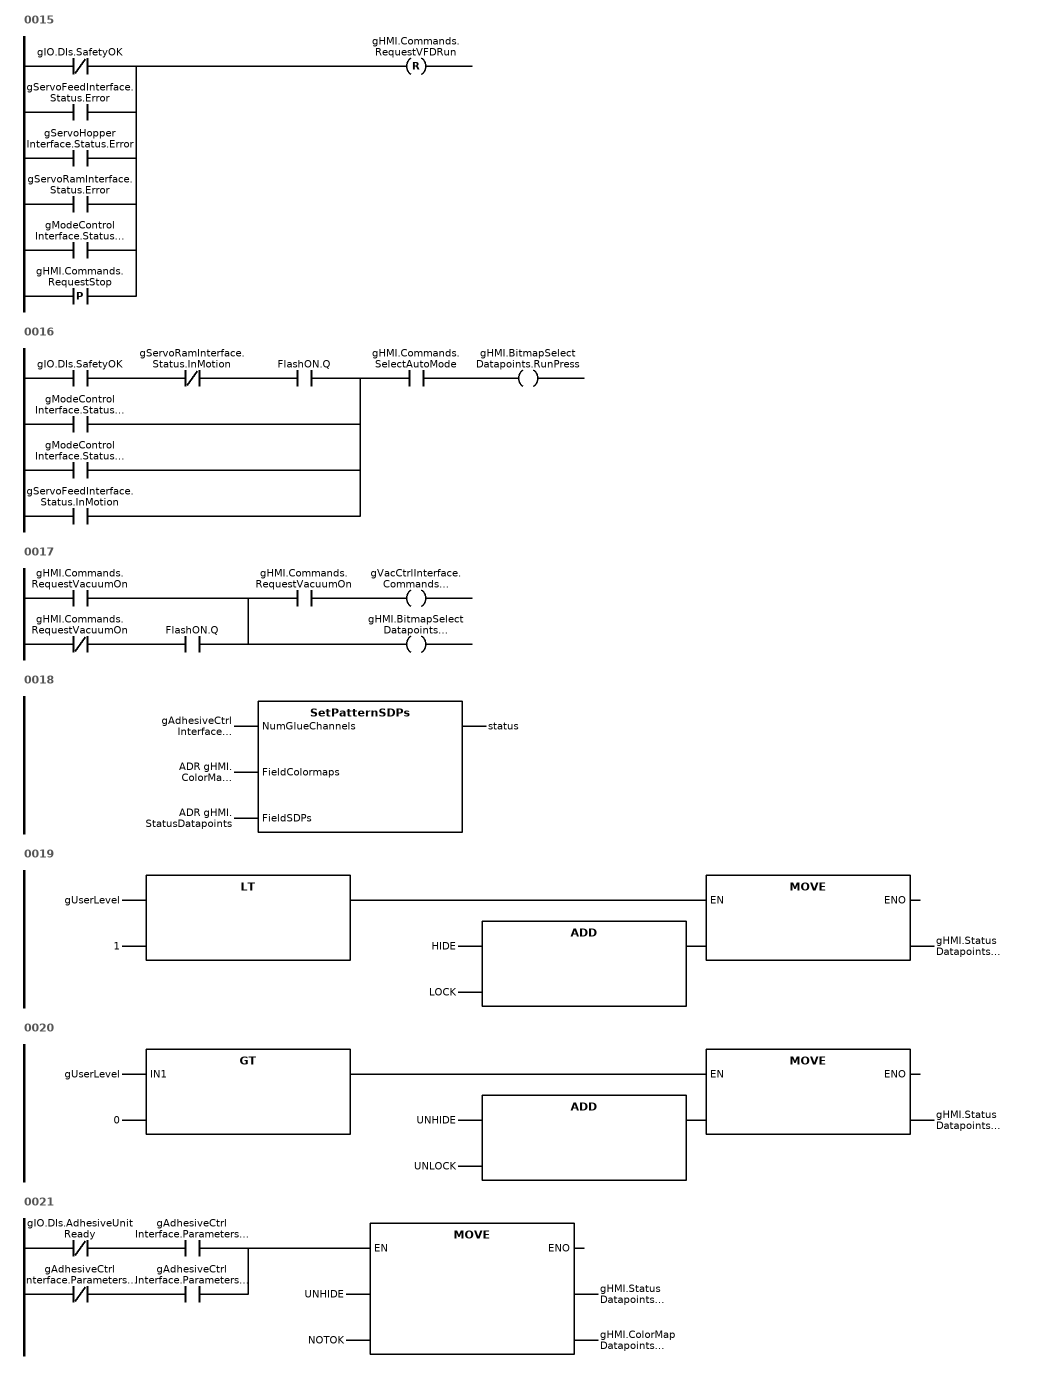
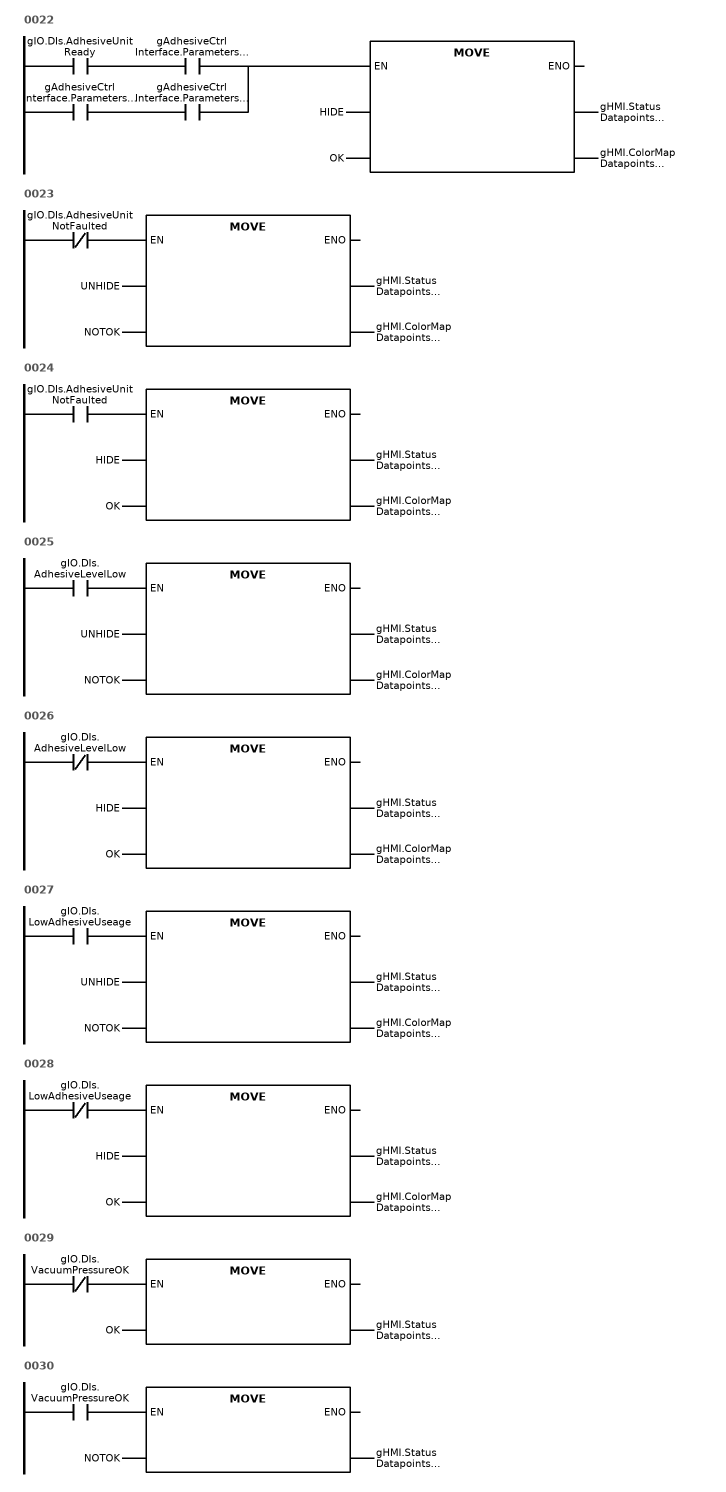
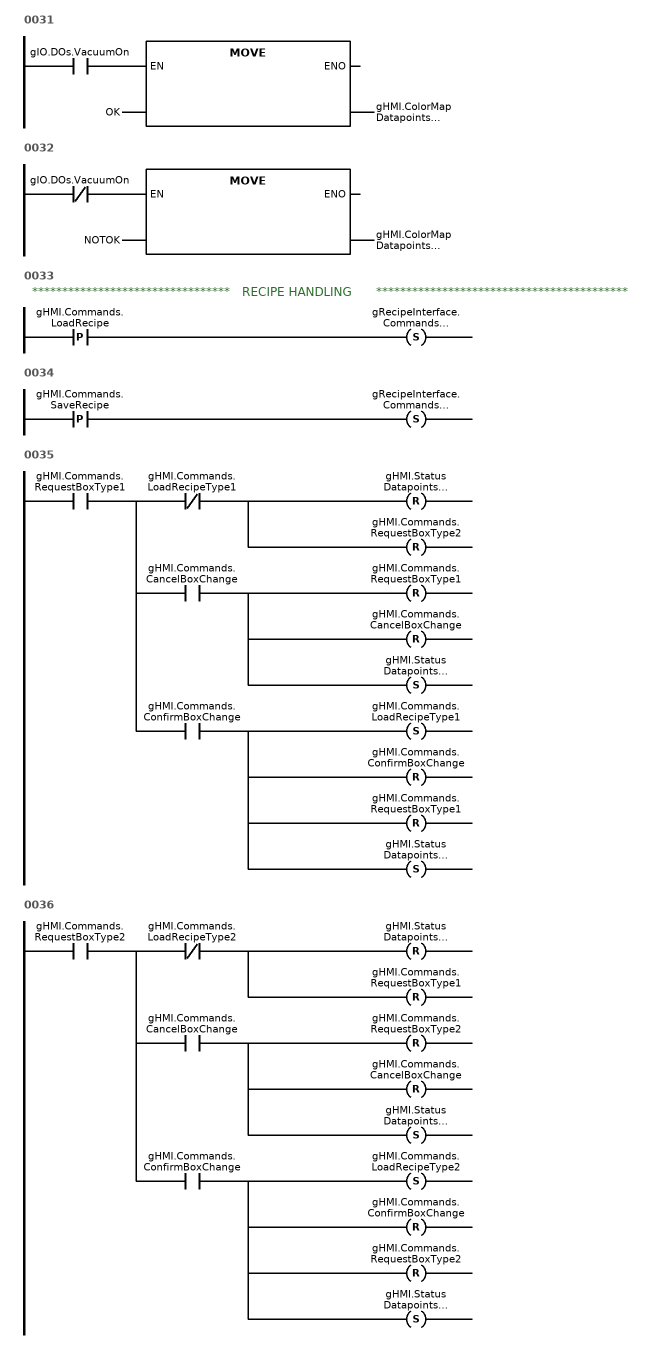
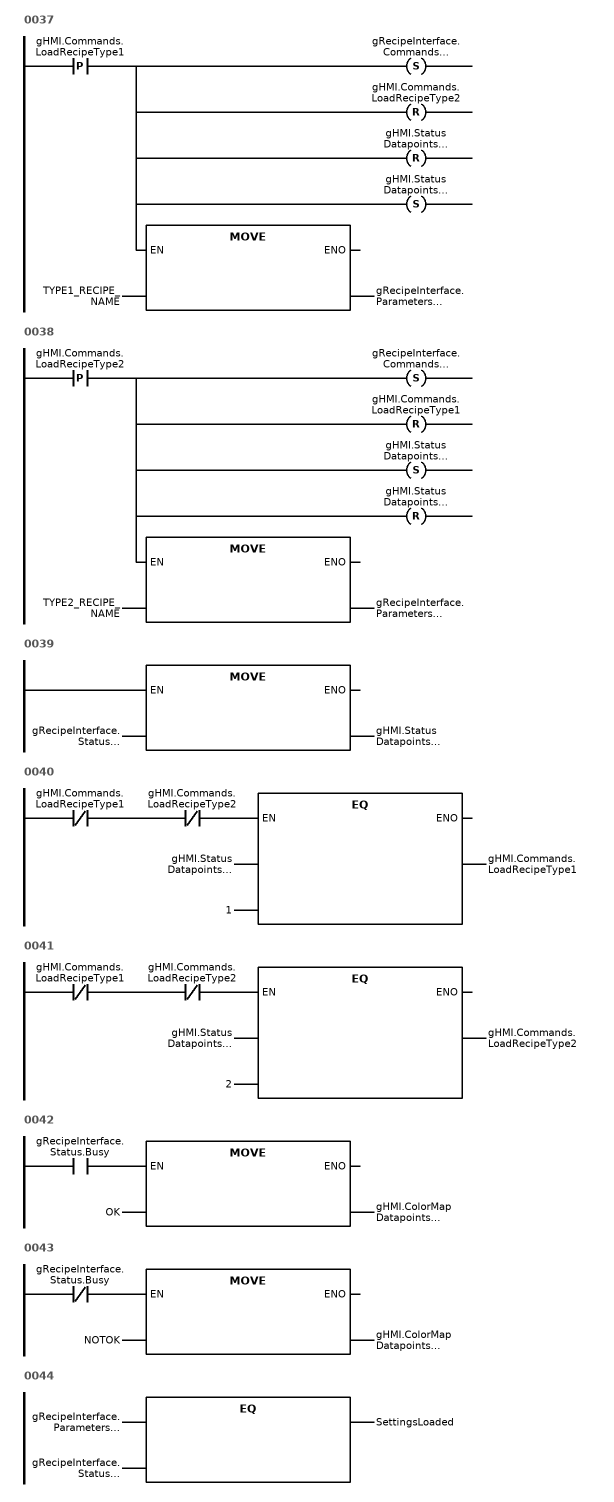
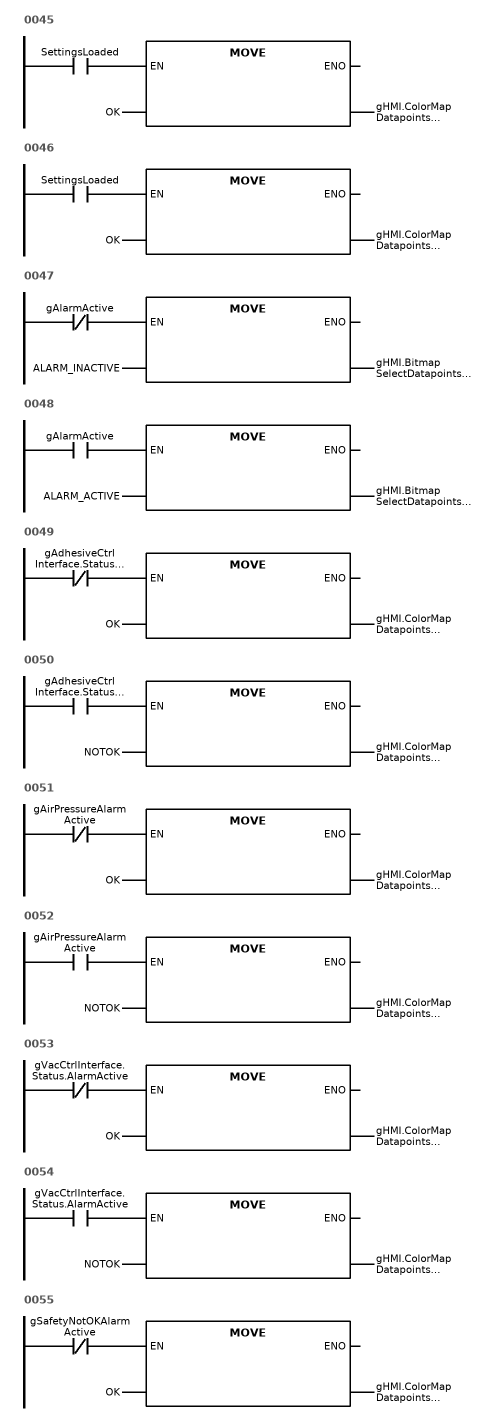
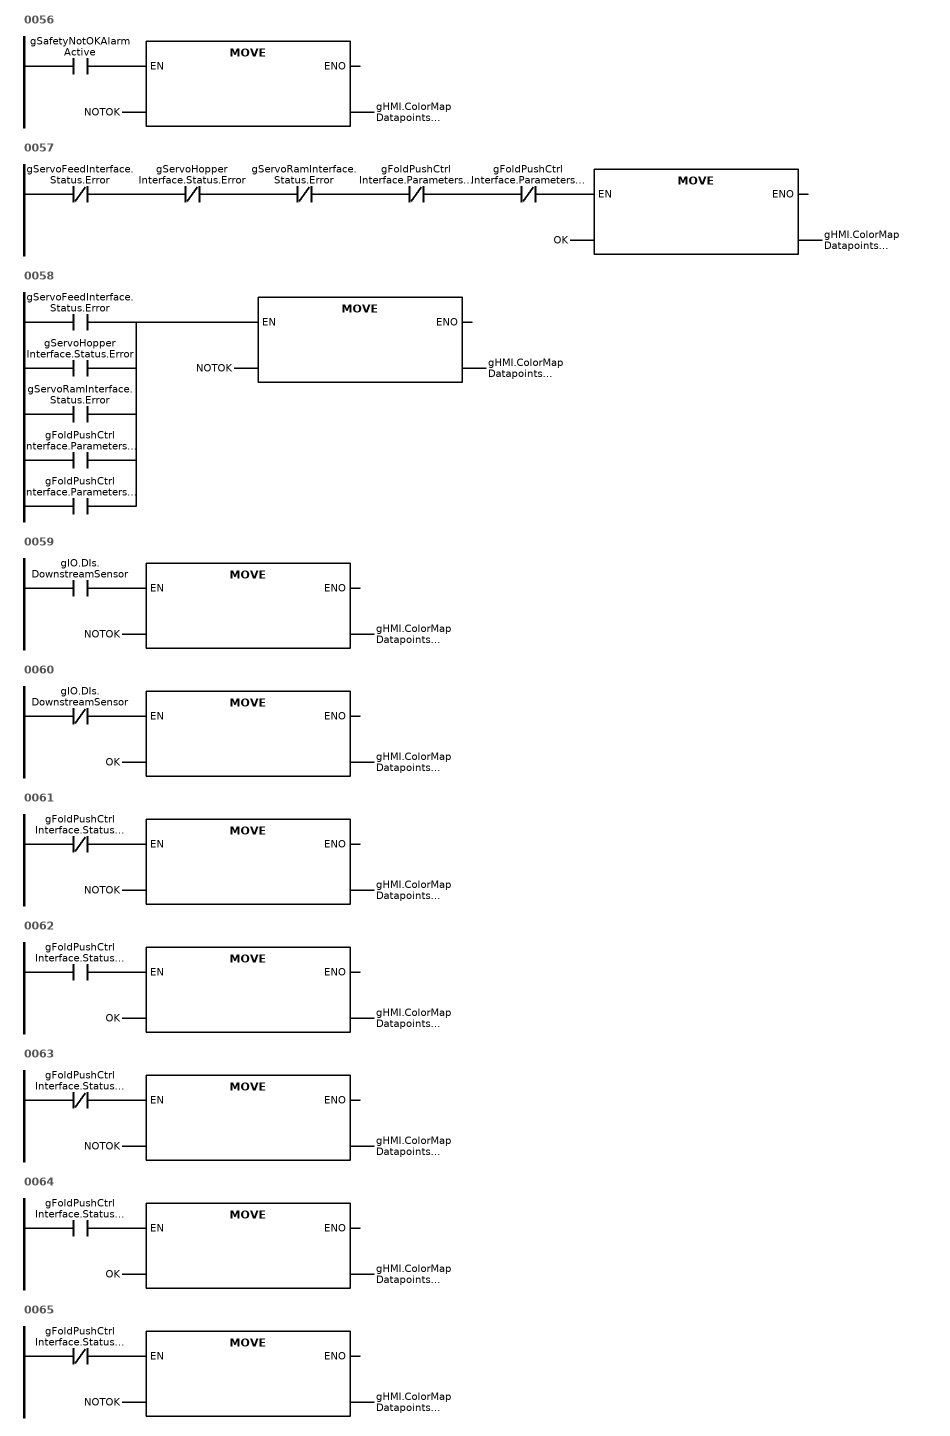
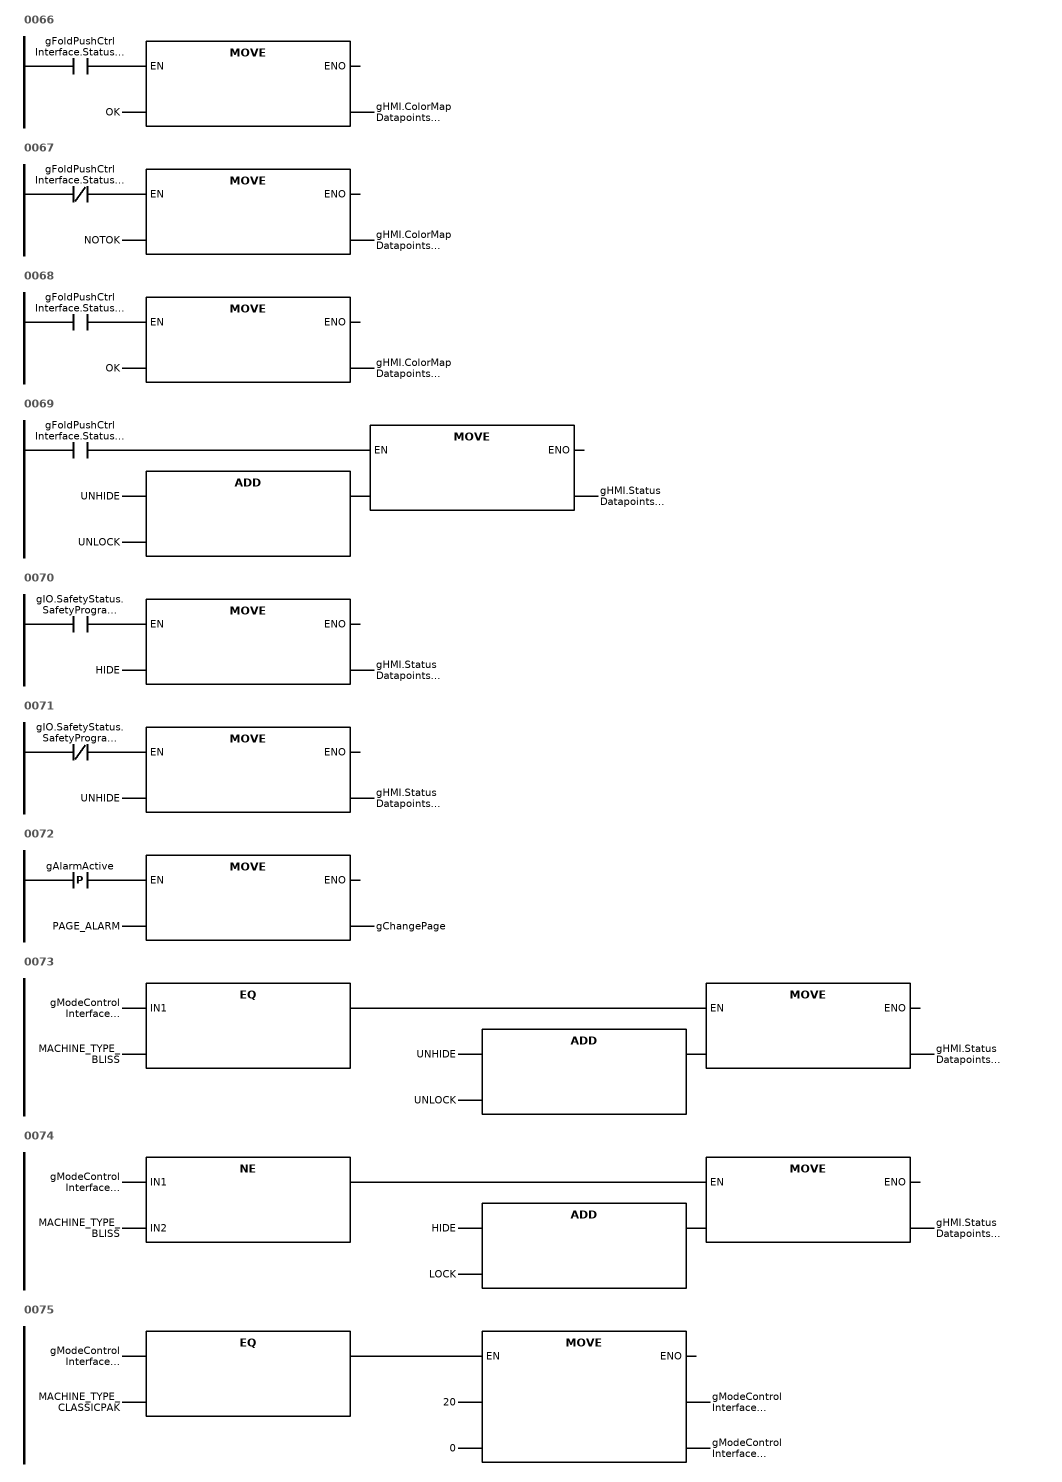
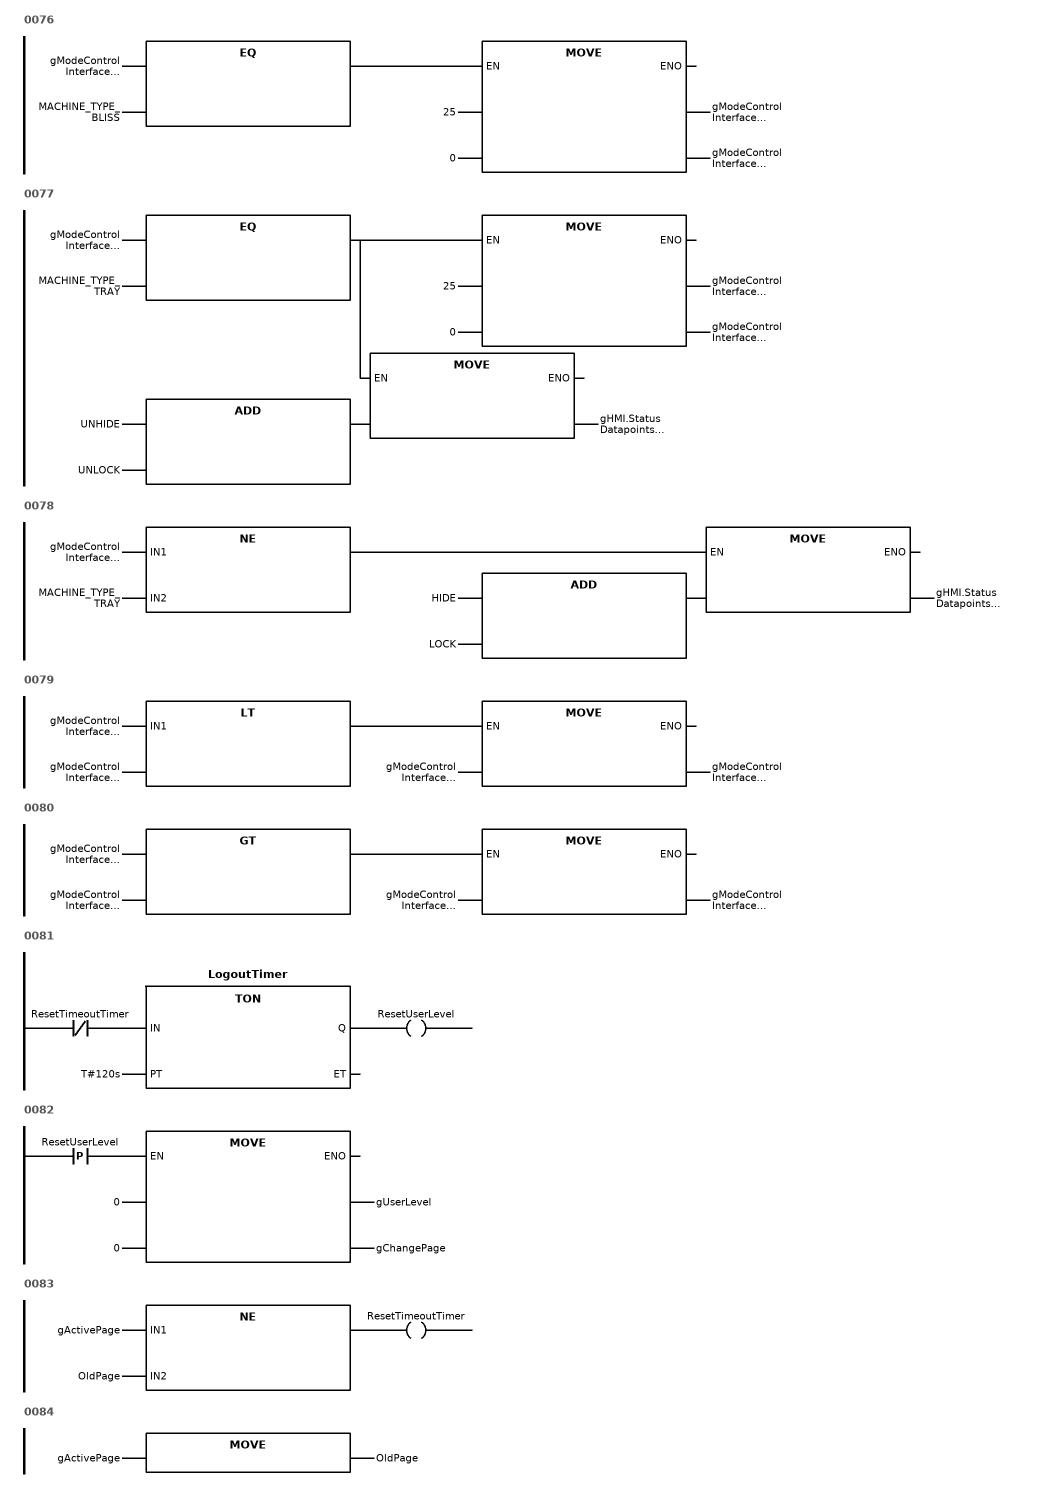
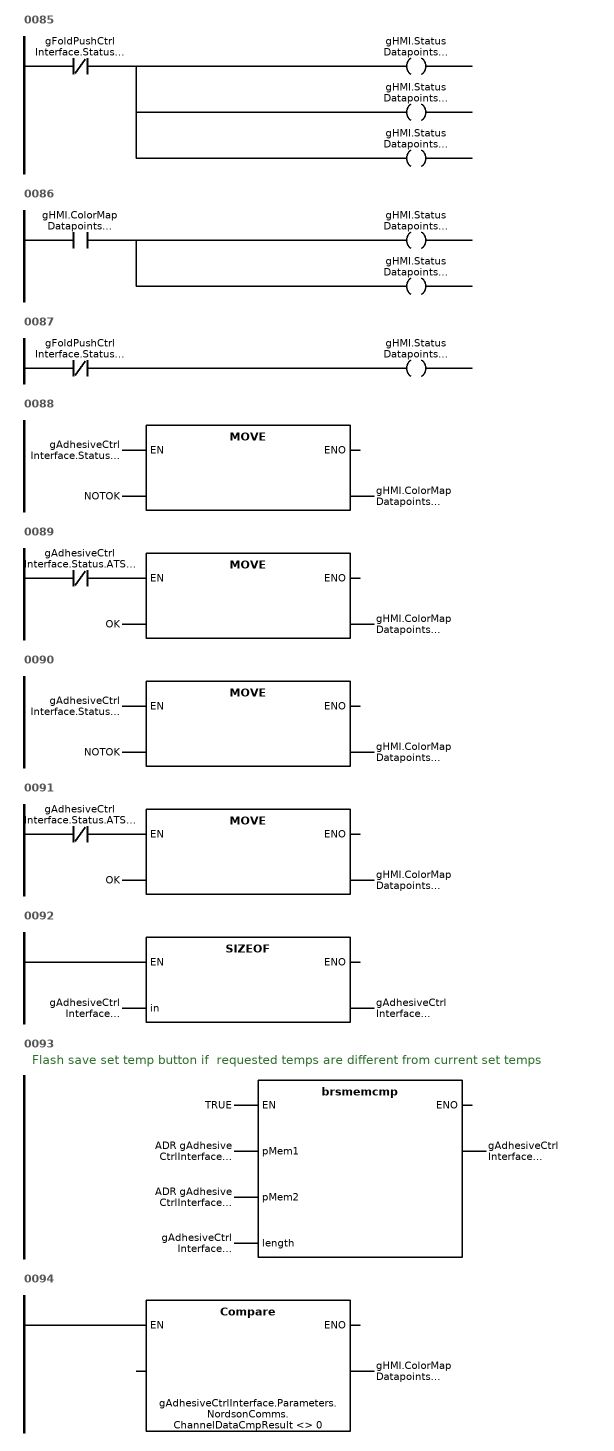
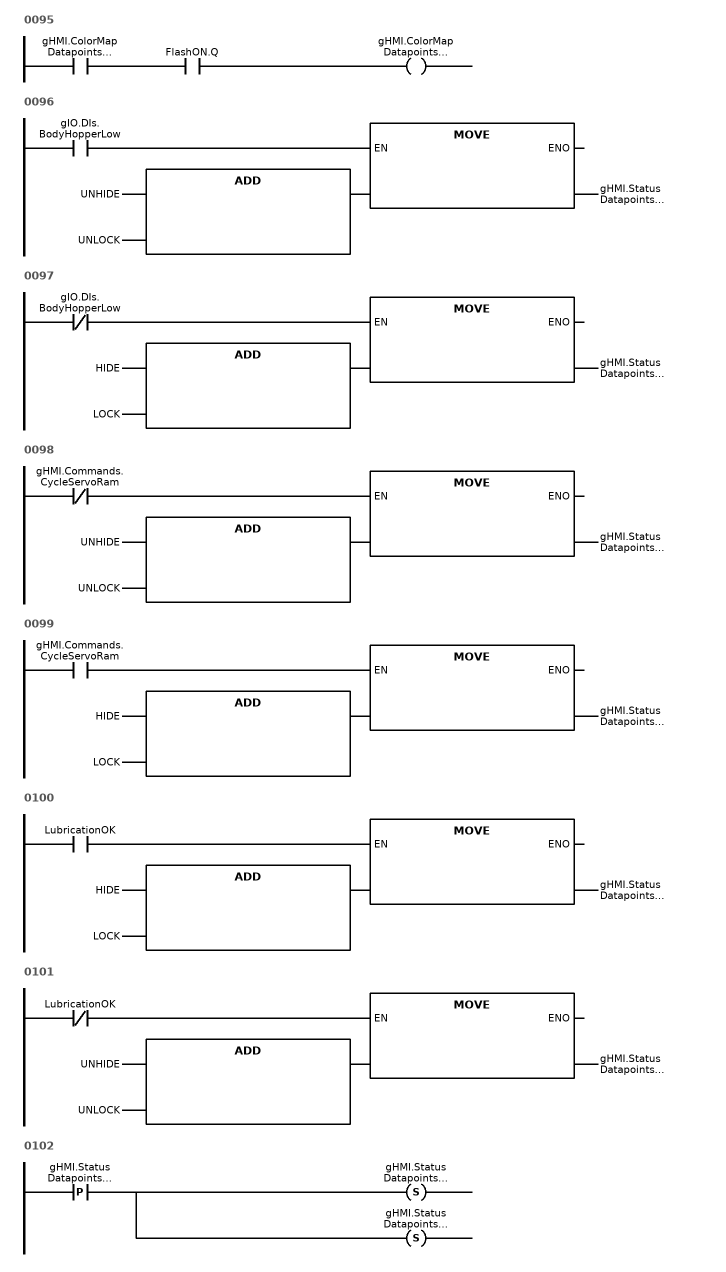
Ladder, written as Structured Text:
```iecst
PROGRAM _CYCLIC
VAR
    _p1 : BOOL;
    _p2 : BOOL;
    _p3 : BOOL;
    _p4 : BOOL;
    _e5 : R_TRIG;
    _p6 : BOOL;
    _p7 : BOOL;
    _p8 : BOOL;
    _p9 : BOOL;
    _e10 : R_TRIG;
    _e11 : R_TRIG;
    _p12 : BOOL;
    _p13 : BOOL;
    _p14 : BOOL;
    _p15 : BOOL;
    _p16 : BOOL;
    _p17 : BOOL;
    _p18 : BOOL;
    _p19 : BOOL;
    _e20 : R_TRIG;
    _e21 : R_TRIG;
    _p22 : BOOL;
    _p23 : BOOL;
    _e24 : R_TRIG;
    _t25 : BOOL;
    _t26 : BOOL;
    _t27 : BOOL;
    _p28 : BOOL;
    _p29 : BOOL;
    _e30 : R_TRIG;
    _p31 : BOOL;
    _p32 : BOOL;
    _p33 : BOOL;
    _e34 : R_TRIG;
END_VAR
(* Network 1 *)
_p1 := gModeControlInterface.Status.BlissPanelAlarmActive;
IF NOT gIO.DIs.SafetyOK OR gServoFeedInterface.Status.Error OR gServoHopperInterface.Status.Error OR gServoRamInterface.Status.Error OR _p1 OR StopFeed OR NOT gServoRamInterface.Status.Homed OR gAlarmActive THEN
    gModeControlInterface.Commands.SetAutoMode := FALSE;
    gModeControlInterface.Commands.SetJogMode := FALSE;
    gHMI.Commands.SelectJogMode := FALSE;
    gHMI.Commands.SelectAutoMode := FALSE;
    gModeControlInterface.Status.Dwelling := FALSE;
END_IF;

(* Network 2 *)
IF NOT gServoRamInterface.Status.Homed THEN gModeControlInterface.Status.Dwelling := FALSE; END_IF;

(* Network 3 *)
IF gHMI.Commands.SelectAutoMode THEN
    gModeControlInterface.Commands.SetAutoMode := TRUE;
    gModeControlInterface.Commands.SetJogMode := FALSE;
END_IF;

(* Network 4 *)
gModeControlInterface.Commands.SetShowMode := gHMI.Commands.EnableShowMode;

(* Network 5 *)
IF gHMI.Commands.SelectJogMode THEN
    gModeControlInterface.Commands.SetJogMode := TRUE;
    gModeControlInterface.Commands.SetAutoMode := FALSE;
    gHMI.Commands.RequestVFDRun := FALSE;
END_IF;

(* Network 6 *)
IF gModeControlInterface.Commands.SetJogMode THEN
    gHMI.ColorMapDatapoints.JogModeSelected := 1;
    gHMI.ColorMapDatapoints.AutoModeSelected := 0;
    gHMI.StatusDatapoints.JogStatusDatapoint := UNHIDE + UNLOCK;
END_IF;

(* Network 7 *)
IF gModeControlInterface.Commands.SetAutoMode THEN
    gHMI.ColorMapDatapoints.JogModeSelected := 0;
    gHMI.ColorMapDatapoints.AutoModeSelected := 1;
    gHMI.StatusDatapoints.JogStatusDatapoint := HIDE + LOCK;
END_IF;

(* Network 8 *)
_p2 := NOT gModeControlInterface.Commands.SetAutoMode AND NOT gModeControlInterface.Commands.SetJogMode;
IF _p2 THEN
    gHMI.ColorMapDatapoints.JogModeSelected := 0;
    gHMI.ColorMapDatapoints.AutoModeSelected := 0;
    gHMI.StatusDatapoints.JogStatusDatapoint := HIDE + LOCK;
END_IF;

(* Network 9 *)
_p3 := gHMI.Commands.SelectAutoMode;
IF _p3 THEN gHMI.StatusDatapoints.AutoModeSDP := UNHIDE + UNLOCK; END_IF;

(* Network 10 *)
_p4 := NOT gHMI.Commands.SelectAutoMode;
IF _p4 THEN gHMI.StatusDatapoints.AutoModeSDP := HIDE + LOCK; END_IF;

(* Network 11: General Lamp Flasher Circuit *)
FlashON(IN := NOT FlashOFF.Q, PT := T#500ms);

(* Network 12: General Lamp Flasher *)
FlashOFF(IN := FlashON.Q, PT := T#500ms);

(* Network 13 *)
gHMI.BitmapSelectDatapoints.ResetPress := (NOT gIO.DIs.SafetyOK AND FlashON.Q) OR gHMI.Commands.RequestReset OR gIO.DIs.SafetyOK;

(* Network 14 *)
gHMI.BitmapSelectDatapoints.StopPress := gHMI.Commands.RequestStop;

(* Network 15 *)
_e5(CLK := gHMI.Commands.RequestStop);
IF NOT gIO.DIs.SafetyOK OR gServoFeedInterface.Status.Error OR gServoHopperInterface.Status.Error OR gServoRamInterface.Status.Error OR gModeControlInterface.Status.BlissPanelAlarmActive OR _e5.Q THEN
    gHMI.Commands.RequestVFDRun := FALSE;
END_IF;

(* Network 16 *)
gHMI.BitmapSelectDatapoints.RunPress := ((gIO.DIs.SafetyOK AND NOT gServoRamInterface.Status.InMotion AND FlashON.Q) OR gModeControlInterface.Status.Dwelling OR gModeControlInterface.Status.WaitingOnDownstream OR gServoFeedInterface.Status.InMotion) AND gHMI.Commands.SelectAutoMode;

(* Network 17 *)
gVacCtrlInterface.Commands.VacuumOn := (gHMI.Commands.RequestVacuumOn OR (NOT gHMI.Commands.RequestVacuumOn AND FlashON.Q)) AND gHMI.Commands.RequestVacuumOn;
gHMI.BitmapSelectDatapoints.VacuumPress := gHMI.Commands.RequestVacuumOn OR (NOT gHMI.Commands.RequestVacuumOn AND FlashON.Q);

(* Network 18 *)
status := SetPatternSDPs(NumGlueChannels := gAdhesiveCtrlInterface.Parameters.NumAdhesiveChannels, FieldColormaps := ADR(gHMI.ColorMapDatapoints), FieldSDPs := ADR(gHMI.StatusDatapoints));

(* Network 19 *)
IF gUserLevel < 1 THEN gHMI.StatusDatapoints.MaintenanceSDP := HIDE + LOCK; END_IF;

(* Network 20 *)
IF gUserLevel > 0 THEN gHMI.StatusDatapoints.MaintenanceSDP := UNHIDE + UNLOCK; END_IF;

(* Network 21 *)
_p6 := NOT gIO.DIs.AdhesiveUnitReady AND gAdhesiveCtrlInterface.Parameters.FeedbackIsHardwire;
_p7 := NOT gAdhesiveCtrlInterface.Parameters.NordsonComms.UnitReady AND gAdhesiveCtrlInterface.Parameters.FeedbackIsModbusTCP;
IF _p6 OR _p7 THEN
    gHMI.StatusDatapoints.AdhesiveUnitNotReadySDP := UNHIDE;
    gHMI.ColorMapDatapoints.AdhesiveUnitReady := NOTOK;
END_IF;

(* Network 22 *)
_p8 := gIO.DIs.AdhesiveUnitReady AND gAdhesiveCtrlInterface.Parameters.FeedbackIsHardwire;
_p9 := gAdhesiveCtrlInterface.Parameters.NordsonComms.UnitReady AND gAdhesiveCtrlInterface.Parameters.FeedbackIsModbusTCP;
IF _p8 OR _p9 THEN
    gHMI.StatusDatapoints.AdhesiveUnitNotReadySDP := HIDE;
    gHMI.ColorMapDatapoints.AdhesiveUnitReady := OK;
END_IF;

(* Network 23 *)
IF NOT gIO.DIs.AdhesiveUnitNotFaulted THEN
    gHMI.StatusDatapoints.AdhesiveUnitFaultSDP := UNHIDE;
    gHMI.ColorMapDatapoints.AdhesiveUnitFault := NOTOK;
END_IF;

(* Network 24 *)
IF gIO.DIs.AdhesiveUnitNotFaulted THEN
    gHMI.StatusDatapoints.AdhesiveUnitFaultSDP := HIDE;
    gHMI.ColorMapDatapoints.AdhesiveUnitFault := OK;
END_IF;

(* Network 25 *)
IF gIO.DIs.AdhesiveLevelLow THEN
    gHMI.StatusDatapoints.AdhesiveUnitLevelLowSDP := UNHIDE;
    gHMI.ColorMapDatapoints.AdhesiveUnitLevelLow := NOTOK;
END_IF;

(* Network 26 *)
IF NOT gIO.DIs.AdhesiveLevelLow THEN
    gHMI.StatusDatapoints.AdhesiveUnitLevelLowSDP := HIDE;
    gHMI.ColorMapDatapoints.AdhesiveUnitLevelLow := OK;
END_IF;

(* Network 27 *)
IF gIO.DIs.LowAdhesiveUseage THEN
    gHMI.StatusDatapoints.AdhesiveUseageLowSDP := UNHIDE;
    gHMI.ColorMapDatapoints.AdhesiveUseageLow := NOTOK;
END_IF;

(* Network 28 *)
IF NOT gIO.DIs.LowAdhesiveUseage THEN
    gHMI.StatusDatapoints.AdhesiveUseageLowSDP := HIDE;
    gHMI.ColorMapDatapoints.AdhesiveUseageLow := OK;
END_IF;

(* Network 29 *)
IF NOT gIO.DIs.VacuumPressureOK THEN gHMI.StatusDatapoints.VacuumPressureFaultSDP := OK; END_IF;

(* Network 30 *)
IF gIO.DIs.VacuumPressureOK THEN gHMI.StatusDatapoints.VacuumPressureFaultSDP := NOTOK; END_IF;

(* Network 31 *)
IF gIO.DOs.VacuumOn THEN gHMI.ColorMapDatapoints.VacuumPumpOn := OK; END_IF;

(* Network 32 *)
IF NOT gIO.DOs.VacuumOn THEN gHMI.ColorMapDatapoints.VacuumPumpOn := NOTOK; END_IF;

(* Network 33: *********************************   RECIPE HANDLING      ****************************************** *)
_e10(CLK := gHMI.Commands.LoadRecipe);
IF _e10.Q THEN gRecipeInterface.Commands.LoadRecipe := TRUE; END_IF;

(* Network 34 *)
_e11(CLK := gHMI.Commands.SaveRecipe);
IF _e11.Q THEN gRecipeInterface.Commands.SaveRecipe := TRUE; END_IF;

(* Network 35 *)
_p12 := gHMI.Commands.RequestBoxType1 AND NOT gHMI.Commands.LoadRecipeType1;
_p13 := gHMI.Commands.RequestBoxType1;
IF _p12 THEN
    gHMI.StatusDatapoints.RecipeDialogSDP.0 := FALSE;
    gHMI.Commands.RequestBoxType2 := FALSE;
END_IF;
_p14 := _p13 AND gHMI.Commands.CancelBoxChange;
IF _p13 AND gHMI.Commands.CancelBoxChange THEN gHMI.Commands.RequestBoxType1 := FALSE; END_IF;
IF _p14 THEN
    gHMI.Commands.CancelBoxChange := FALSE;
    gHMI.StatusDatapoints.RecipeDialogSDP.0 := TRUE;
END_IF;
_p15 := _p13 AND gHMI.Commands.ConfirmBoxChange;
IF _p13 AND gHMI.Commands.ConfirmBoxChange THEN gHMI.Commands.LoadRecipeType1 := TRUE; END_IF;
IF _p15 THEN
    gHMI.Commands.ConfirmBoxChange := FALSE;
    gHMI.Commands.RequestBoxType1 := FALSE;
    gHMI.StatusDatapoints.RecipeDialogSDP.0 := TRUE;
END_IF;

(* Network 36 *)
_p16 := gHMI.Commands.RequestBoxType2 AND NOT gHMI.Commands.LoadRecipeType2;
_p17 := gHMI.Commands.RequestBoxType2;
IF _p16 THEN
    gHMI.StatusDatapoints.RecipeDialogSDP.0 := FALSE;
    gHMI.Commands.RequestBoxType1 := FALSE;
END_IF;
_p18 := _p17 AND gHMI.Commands.CancelBoxChange;
IF _p17 AND gHMI.Commands.CancelBoxChange THEN gHMI.Commands.RequestBoxType2 := FALSE; END_IF;
IF _p18 THEN
    gHMI.Commands.CancelBoxChange := FALSE;
    gHMI.StatusDatapoints.RecipeDialogSDP.0 := TRUE;
END_IF;
_p19 := _p17 AND gHMI.Commands.ConfirmBoxChange;
IF _p17 AND gHMI.Commands.ConfirmBoxChange THEN gHMI.Commands.LoadRecipeType2 := TRUE; END_IF;
IF _p19 THEN
    gHMI.Commands.ConfirmBoxChange := FALSE;
    gHMI.Commands.RequestBoxType2 := FALSE;
    gHMI.StatusDatapoints.RecipeDialogSDP.0 := TRUE;
END_IF;

(* Network 37 *)
_e20(CLK := gHMI.Commands.LoadRecipeType1);
IF _e20.Q THEN
    gRecipeInterface.Commands.LoadRecipe := TRUE;
    gHMI.Commands.LoadRecipeType2 := FALSE;
    gHMI.StatusDatapoints.RecipeReq2SDP.1 := FALSE;
    gHMI.StatusDatapoints.RecipeReq1SDP.1 := TRUE;
    gRecipeInterface.Parameters.RecipeName := TYPE1_RECIPE_NAME;
END_IF;

(* Network 38 *)
_e21(CLK := gHMI.Commands.LoadRecipeType2);
IF _e21.Q THEN
    gRecipeInterface.Commands.LoadRecipe := TRUE;
    gHMI.Commands.LoadRecipeType1 := FALSE;
    gHMI.StatusDatapoints.RecipeReq2SDP.1 := TRUE;
    gHMI.StatusDatapoints.RecipeReq1SDP.1 := FALSE;
    gRecipeInterface.Parameters.RecipeName := TYPE2_RECIPE_NAME;
END_IF;

(* Network 39 *)
gHMI.StatusDatapoints.RecipeIndexSDP := gRecipeInterface.Status.LoadedRecipeIndex;

(* Network 40 *)
_p22 := NOT gHMI.Commands.LoadRecipeType1 AND NOT gHMI.Commands.LoadRecipeType2;
IF _p22 THEN gHMI.Commands.LoadRecipeType1 := gHMI.StatusDatapoints.RecipeIndexSDP = 1; END_IF;

(* Network 41 *)
_p23 := NOT gHMI.Commands.LoadRecipeType1 AND NOT gHMI.Commands.LoadRecipeType2;
IF _p23 THEN gHMI.Commands.LoadRecipeType2 := gHMI.StatusDatapoints.RecipeIndexSDP = 2; END_IF;

(* Network 42 *)
IF gRecipeInterface.Status.Busy THEN gHMI.ColorMapDatapoints.RecipeSystemBusy := OK; END_IF;

(* Network 43 *)
IF NOT gRecipeInterface.Status.Busy THEN gHMI.ColorMapDatapoints.RecipeSystemBusy := NOTOK; END_IF;

(* Network 44 *)
SettingsLoaded := gRecipeInterface.Parameters.RecipeName = gRecipeInterface.Status.LoadedRecipeName;

(* Network 45 *)
IF SettingsLoaded THEN gHMI.ColorMapDatapoints.RecipeLoaded := OK; END_IF;

(* Network 46 *)
IF SettingsLoaded THEN gHMI.ColorMapDatapoints.RecipeLoaded := OK; END_IF;

(* Network 47 *)
IF NOT gAlarmActive THEN gHMI.BitmapSelectDatapoints.AlarmActive := ALARM_INACTIVE; END_IF;

(* Network 48 *)
IF gAlarmActive THEN gHMI.BitmapSelectDatapoints.AlarmActive := ALARM_ACTIVE; END_IF;

(* Network 49 *)
IF NOT gAdhesiveCtrlInterface.Status.AlarmActive THEN
    gHMI.ColorMapDatapoints.AdhesiveSystemOK := OK;
END_IF;

(* Network 50 *)
IF gAdhesiveCtrlInterface.Status.AlarmActive THEN
    gHMI.ColorMapDatapoints.AdhesiveSystemOK := NOTOK;
END_IF;

(* Network 51 *)
IF NOT gAirPressureAlarmActive THEN gHMI.ColorMapDatapoints.AirPressureOK := OK; END_IF;

(* Network 52 *)
IF gAirPressureAlarmActive THEN gHMI.ColorMapDatapoints.AirPressureOK := NOTOK; END_IF;

(* Network 53 *)
IF NOT gVacCtrlInterface.Status.AlarmActive THEN gHMI.ColorMapDatapoints.VacuumOK := OK; END_IF;

(* Network 54 *)
IF gVacCtrlInterface.Status.AlarmActive THEN gHMI.ColorMapDatapoints.VacuumOK := NOTOK; END_IF;

(* Network 55 *)
IF NOT gSafetyNotOKAlarmActive THEN gHMI.ColorMapDatapoints.SafetyOK := OK; END_IF;

(* Network 56 *)
IF gSafetyNotOKAlarmActive THEN gHMI.ColorMapDatapoints.SafetyOK := NOTOK; END_IF;

(* Network 57 *)
IF NOT gServoFeedInterface.Status.Error AND NOT gServoHopperInterface.Status.Error AND NOT gServoRamInterface.Status.Error AND NOT gFoldPushCtrlInterface.Parameters.LinMotBotFolder.Status.Error AND NOT gFoldPushCtrlInterface.Parameters.LinMotTopFolder.Status.Error THEN
    gHMI.ColorMapDatapoints.DriveFaultOK := OK;
END_IF;

(* Network 58 *)
IF gServoFeedInterface.Status.Error OR gServoHopperInterface.Status.Error OR gServoRamInterface.Status.Error OR gFoldPushCtrlInterface.Parameters.LinMotBotFolder.Status.Error OR gFoldPushCtrlInterface.Parameters.LinMotTopFolder.Status.Error THEN
    gHMI.ColorMapDatapoints.DriveFaultOK := NOTOK;
END_IF;

(* Network 59 *)
IF gIO.DIs.DownstreamSensor THEN gHMI.ColorMapDatapoints.DownstreamSensorOK := NOTOK; END_IF;

(* Network 60 *)
IF NOT gIO.DIs.DownstreamSensor THEN gHMI.ColorMapDatapoints.DownstreamSensorOK := OK; END_IF;

(* Network 61 *)
IF NOT gFoldPushCtrlInterface.Status.TopFoldValveStatus THEN
    gHMI.ColorMapDatapoints.Valve1OK := NOTOK;
END_IF;

(* Network 62 *)
IF gFoldPushCtrlInterface.Status.TopFoldValveStatus THEN gHMI.ColorMapDatapoints.Valve1OK := OK; END_IF;

(* Network 63 *)
IF NOT gFoldPushCtrlInterface.Status.BottomFoldValveStatus THEN
    gHMI.ColorMapDatapoints.Valve2OK := NOTOK;
END_IF;

(* Network 64 *)
IF gFoldPushCtrlInterface.Status.BottomFoldValveStatus THEN
    gHMI.ColorMapDatapoints.Valve2OK := OK;
END_IF;

(* Network 65 *)
IF NOT gFoldPushCtrlInterface.Status.CompOnValveStatus THEN
    gHMI.ColorMapDatapoints.Valve3OK := NOTOK;
END_IF;

(* Network 66 *)
IF gFoldPushCtrlInterface.Status.CompOnValveStatus THEN gHMI.ColorMapDatapoints.Valve3OK := OK; END_IF;

(* Network 67 *)
IF NOT gFoldPushCtrlInterface.Status.PushValveStatus THEN
    gHMI.ColorMapDatapoints.Valve4OK := NOTOK;
END_IF;

(* Network 68 *)
IF gFoldPushCtrlInterface.Status.PushValveStatus THEN gHMI.ColorMapDatapoints.Valve4OK := OK; END_IF;

(* Network 69 *)
IF gFoldPushCtrlInterface.Status.HardwireConfig THEN
    gHMI.StatusDatapoints.HardwireValveSDP := UNHIDE + UNLOCK;
END_IF;

(* Network 70 *)
IF gIO.SafetyStatus.SafetyProgramRunning THEN gHMI.StatusDatapoints.SafetyStartingSDP := HIDE; END_IF;

(* Network 71 *)
IF NOT gIO.SafetyStatus.SafetyProgramRunning THEN
    gHMI.StatusDatapoints.SafetyStartingSDP := UNHIDE;
END_IF;

(* Network 72 *)
_e24(CLK := gAlarmActive);
IF _e24.Q THEN gChangePage := PAGE_ALARM; END_IF;

(* Network 73 *)
IF gModeControlInterface.Parameters.MachineType = MACHINE_TYPE_BLISS THEN
    gHMI.StatusDatapoints.BlissSDP := UNHIDE + UNLOCK;
END_IF;

(* Network 74 *)
IF gModeControlInterface.Parameters.MachineType <> MACHINE_TYPE_BLISS THEN
    gHMI.StatusDatapoints.BlissSDP := HIDE + LOCK;
END_IF;

(* Network 75 *)
_t25 := gModeControlInterface.Parameters.MachineType = MACHINE_TYPE_CLASSICPAK;
IF _t25 THEN
    gModeControlInterface.Parameters.MaxPPM := 20;
    gModeControlInterface.Parameters.MinPPM := 0;
END_IF;

(* Network 76 *)
_t26 := gModeControlInterface.Parameters.MachineType = MACHINE_TYPE_BLISS;
IF _t26 THEN
    gModeControlInterface.Parameters.MaxPPM := 25;
    gModeControlInterface.Parameters.MinPPM := 0;
END_IF;

(* Network 77 *)
_t27 := gModeControlInterface.Parameters.MachineType = MACHINE_TYPE_TRAY;
IF _t27 THEN
    gModeControlInterface.Parameters.MaxPPM := 25;
    gModeControlInterface.Parameters.MinPPM := 0;
    gHMI.StatusDatapoints.TraySDP := UNHIDE + UNLOCK;
END_IF;

(* Network 78 *)
IF gModeControlInterface.Parameters.MachineType <> MACHINE_TYPE_TRAY THEN
    gHMI.StatusDatapoints.TraySDP := HIDE + LOCK;
END_IF;

(* Network 79 *)
_p28 := gModeControlInterface.Parameters.MaxPPM < gModeControlInterface.Parameters.PiecesPerMinute;
IF _p28 THEN
    gModeControlInterface.Parameters.PiecesPerMinute := gModeControlInterface.Parameters.MaxPPM;
END_IF;

(* Network 80 *)
_p29 := gModeControlInterface.Parameters.MinPPM > gModeControlInterface.Parameters.PiecesPerMinute;
IF _p29 THEN
    gModeControlInterface.Parameters.PiecesPerMinute := gModeControlInterface.Parameters.MinPPM;
END_IF;

(* Network 81 *)
LogoutTimer(IN := NOT ResetTimeoutTimer, PT := T#120s);
ResetUserLevel := LogoutTimer.Q;

(* Network 82 *)
_e30(CLK := ResetUserLevel);
IF _e30.Q THEN
    gUserLevel := 0;
    gChangePage := 0;
END_IF;

(* Network 83 *)
ResetTimeoutTimer := gActivePage <> OldPage;

(* Network 84 *)
OldPage := gActivePage;

(* Network 85 *)
gHMI.StatusDatapoints.LinMotSDP.0 := NOT gFoldPushCtrlInterface.Status.LinMotConfig;
gHMI.StatusDatapoints.LinMotTopHomeSDP.0 := NOT gFoldPushCtrlInterface.Status.LinMotConfig;
gHMI.StatusDatapoints.LinMotBotHomeSDP.0 := NOT gFoldPushCtrlInterface.Status.LinMotConfig;

(* Network 86 *)
_p31 := gHMI.ColorMapDatapoints.AutoModeSelected.0;
gHMI.StatusDatapoints.LinMotTopHomeSDP.1 := gHMI.ColorMapDatapoints.AutoModeSelected.0;
gHMI.StatusDatapoints.LinMotBotHomeSDP.1 := _p31;

(* Network 87 *)
gHMI.StatusDatapoints.PnuematicFolderSDP.0 := NOT gFoldPushCtrlInterface.Status.PneumaticConfig;

(* Network 88 *)
IF gAdhesiveCtrlInterface.Status.ATS_AddOnOverLimit THEN
    gHMI.ColorMapDatapoints.ATSAddOnOver := NOTOK;
END_IF;

(* Network 89 *)
IF NOT gAdhesiveCtrlInterface.Status.ATS_AddOnOverLimit THEN
    gHMI.ColorMapDatapoints.ATSAddOnOver := OK;
END_IF;

(* Network 90 *)
IF gAdhesiveCtrlInterface.Status.ATS_AddOnUnderLimit THEN
    gHMI.ColorMapDatapoints.ATSAddOnUnder := NOTOK;
END_IF;

(* Network 91 *)
IF NOT gAdhesiveCtrlInterface.Status.ATS_AddOnUnderLimit THEN
    gHMI.ColorMapDatapoints.ATSAddOnUnder := OK;
END_IF;

(* Network 92 *)
gAdhesiveCtrlInterface.Parameters.NordsonComms.ChannelDataSize := SIZEOF(in := gAdhesiveCtrlInterface.Parameters.NordsonComms.ChannelSetTempActual);

(* Network 93: Flash save set temp button if  requested temps are different from current set temps *)
gAdhesiveCtrlInterface.Parameters.NordsonComms.ChannelDataCmpResult := brsmemcmp(pMem1 := ADR(gAdhesiveCtrlInterface.Parameters.NordsonComms.ChannelSetTempActual), pMem2 := ADR(gAdhesiveCtrlInterface.Parameters.NordsonComms.ChannelSetTempRequested), length := gAdhesiveCtrlInterface.Parameters.NordsonComms.ChannelDataSize);

(* Network 94 *)
gHMI.ColorMapDatapoints.NordsonEditTemps := gAdhesiveCtrlInterface.Parameters.NordsonComms.ChannelDataCmpResult <> 0;

(* Network 95 *)
gHMI.ColorMapDatapoints.NordsonEditTemps.0 := gHMI.ColorMapDatapoints.NordsonEditTemps.0 AND FlashON.Q;

(* Network 96 *)
IF gIO.DIs.BodyHopperLow THEN gHMI.StatusDatapoints.HopperLowSDP := UNHIDE + UNLOCK; END_IF;

(* Network 97 *)
IF NOT gIO.DIs.BodyHopperLow THEN gHMI.StatusDatapoints.HopperLowSDP := HIDE + LOCK; END_IF;

(* Network 98 *)
_p32 := NOT gHMI.Commands.CycleServoRam;
IF _p32 THEN gHMI.StatusDatapoints.HomeServoRamSDP := UNHIDE + UNLOCK; END_IF;

(* Network 99 *)
_p33 := gHMI.Commands.CycleServoRam;
IF _p33 THEN gHMI.StatusDatapoints.HomeServoRamSDP := HIDE + LOCK; END_IF;

(* Network 100 *)
IF LubricationOK THEN gHMI.StatusDatapoints.LubeSDP := HIDE + LOCK; END_IF;

(* Network 101 *)
IF NOT LubricationOK THEN gHMI.StatusDatapoints.LubeSDP := UNHIDE + UNLOCK; END_IF;

(* Network 102 *)
_e34(CLK := gHMI.StatusDatapoints.AdhesivePatternConfirmedSDP.0);
IF _e34.Q THEN
    gHMI.StatusDatapoints.AdhesivePatternConfirmDialogSDP.0 := TRUE;
    gHMI.StatusDatapoints.AdhesivePatternDialogSDP.0 := TRUE;
END_IF;
END_PROGRAM
```

#### Init.st
```iecst
PROGRAM _INIT

	gActivePage; //useonce in code so that HMI can see this variable

//	gHMI.ColorMapDatapoints.AirPressureOK := OK;
//	gHMI.ColorMapDatapoints.SafetyOK := OK;
	//	gHMI.ColorMapDatapoints.colorma
	gHMI.StatusDatapoints.SmartVacuumLayerSDP := HIDE + LOCK;
	gHMI.StatusDatapoints.ServoLayerSDP := HIDE + LOCK;

	gHMI.ColorMapDatapoints.AdhesiveUnitServiceNeeded := OK;

	gModeControlInterface.Parameters.MaxPPM := 20; //set the max ppm to the smallest max that you'd see for any machine type. We think we can get into a state where the set PPM is put to 0 on startup if this number is 0

	gHMI.StatusDatapoints.RecipeDialogSDP := HIDE;

END_PROGRAM
```

- Visualisation Logical/HMI/Visu (not shown)

- Project.language (not shown)

### Program Logical/ncsdcctrl (IEC)

#### ncsdcctrlCyclic.st
```iecst
PROGRAM _CYCLIC

(* ### BEGIN gRamAxis ### *)

(* life counter emulation of digital inputs *)
    gRamAxis_DiDoIf.iLifeCntReference := gRamAxis_DiDoIf.iLifeCntReference + 1;
    gRamAxis_DiDoIf.iLifeCntNegHwEnd  := gRamAxis_DiDoIf.iLifeCntNegHwEnd  + 1;
	gRamAxis_DiDoIf.iLifeCntPosHwEnd  := gRamAxis_DiDoIf.iLifeCntPosHwEnd  + 1;
//	gRamAxis_EncIf16.iLifeCnt := gRamAxis_EncIf16.iLifeCnt + 1;

//	gRamAxis_EncIf16.iActPos := UDINT_TO_INT(gIO.Encoders.SickSSIPos);

(* ### END gRamAxis ### *)

END_PROGRAM
```

#### ncsdcctrlInit.st
```iecst
PROGRAM _INIT

(* ### BEGIN gRamAxis ### *)

(* initialize variables *)
	gRamAxis_HW.DrvIf_Typ := ncSDC_DRVSERVO16;
	brsstrcpy( ADR(gRamAxis_HW.DrvIf_Name[0]), ADR('gRamAxis_DrvIf') );
//	gRamAxis_HW.EncIf1_Typ := ncSDC_ENC16;
//	brsstrcpy( ADR(gRamAxis_HW.EncIf1_Name), ADR('gRamAxis_EncIf16') );
	gRamAxis_HW.DiDoIf_Typ := ncSDC_DIDO;
	brsstrcpy( ADR(gRamAxis_HW.DiDoIf_Name[0]), ADR('gRamAxis_DiDoIf') );

	(* force variable offset generation *)
	gRamAxis.size                      := gRamAxis.size;
	gRamAxis_DrvIf.iLifeCnt            := gRamAxis_DrvIf.iLifeCnt;
	gRamAxis_DiDoIf.iLifeCntDriveReady := gRamAxis_DiDoIf.iLifeCntDriveReady;
	gRamAxis_ModuleOk                  := gRamAxis_ModuleOk;

	(* assign your hardware inputs here*)

	(*      gRamAxis_DiDoIf.iPosHwEnd  := gRamAxis_DiDoIf.iPosHwEnd;
	gRamAxis_DiDoIf.iNegHwEnd  := gRamAxis_DiDoIf.iNegHwEnd;
	gRamAxis_DiDoIf.iReference := gRamAxis_DiDoIf.iReference;
	*)

	(* ### END gRamAxis ### *)

END_PROGRAM
```

### Program Logical/EncoderDecoding (ANSIC)

#### Cyclic.c - Cyclic code
```c
#include <bur/plctypes.h>

#ifdef _DEFAULT_INCLUDES
	#include <AsDefault.h>
#endif

void _CYCLIC ProgramCyclic(void)
{
	/*
	BitPackedGrayCode = 0;

	for (i = 0; i < 16; i++)
	{
		BitPackedGrayCode = BitPackedGrayCode | (gIO.DIs.SSI_Parallel.Bits[i] << i);
	}
*/

	//	EncoderPos = grayToBinary(BitPackedGrayCode);

	//num = grayCodeBitPacker(gIO.DIs.SSI_Parallel.Bits);

		EncoderPos = grayToBinary(gIO.DIs.SSI_Parallel.Bits);

}
```

#### Variables.var - Local variables
```iecst
VAR
	num : UDINT;
	EncoderPos : UDINT;
	BitPackedGrayCode : UDINT;
	i : UINT;
END_VAR
```

### Program Logical/Stacklight/PatliteComm (IEC) - Patlite Modbus Comm Program

#### Patelite.st - Stacklight control code for Patlite LA6
```iecst
PROGRAM _INIT

	(* init values *)
	mb_station 			:= 'IF2.ST3';					(* path to modbus station *)
	//This is a new Line3

END_PROGRAM

PROGRAM _CYCLIC

	IF gIsSimulated = FALSE THEN
		//Patlight comms forced to idle state if light stack type is not PATLITE
		IF(gModeControlInterface.Parameters.LightStackSelection <> LIGHTSTACK_PATLITE) THEN
			ErrorCount := 0;
			CommState := PATLITE_STATE_STANDBY;
			CurrentLightGroup := GROUP_1_POWER_ON;

		END_IF

		CASE (CommState) OF

			(***************** PATLITE_STATE STANDBY: CHECK THE MACHINE PATLITE_STATE TO SET LIGHT MODE ***************************)
			PATLITE_STATE_STANDBY:

				(*Check conditions for the light group *)
				IF NOT(gIO.DIs.SafetyOK) THEN
					NextLightGroup := GROUP_5_SAFETY;

				ELSIF gHMI.BitmapSelectDatapoints.RunPress THEN
					NextLightGroup := GROUP_4_RUN;

				ELSIF (gIO.DIs.AirPressureOK AND gAdhesiveCtrlInterface.Status.UnitReady) THEN
					NextLightGroup := GROUP_3_HEAT_AIR_OK;

				ELSE
					NextLightGroup := GROUP_2_HEATING;

				END_IF

				(*If the light group changes, go to the write registry state*)
				IF NextLightGroup <> CurrentLightGroup THEN
					CurrentLightGroup := NextLightGroup;
					CommState := PATLITE_STATE_WRITE_REGISTER;

				END_IF

				IF(gModeControlInterface.Parameters.LightStackSelection <> LIGHTSTACK_PATLITE) THEN
					ErrorCount := 0;
					CommState := PATLITE_STATE_STANDBY;
				END_IF

			(***************** PATLITE_STATE WRITE REGISTER: WRITE THE STACKLIGHT REGISTER TO SET LIGHT MODE ***************************)
			PATLITE_STATE_WRITE_REGISTER:

				mbWriteSingleRegister_0.enable 			:= 1;
				mbWriteSingleRegister_0.pStation 		:= ADR(mb_station);
				mbWriteSingleRegister_0.startAddress 	:= GROUP_REG_ADR;
				mbWriteSingleRegister_0.value 			:= DINT_TO_UINT(CurrentLightGroup) + GROUP_OFFSET;
				mbWriteSingleRegister_0();										(* call function block *)
				IF (mbWriteSingleRegister_0.status <> ERR_FUB_BUSY) THEN
					IF mbWriteSingleRegister_0.status = 0 THEN
						(*Successful write, go to standby*)
						CommState := PATLITE_STATE_STANDBY;
						CommError := FALSE;
						ErrorCount := 0;
					ELSE
						(*Error writing, go to error state*)
						CommState := PATLITE_STATE_ERROR;
						ErrorCount := ErrorCount+1;
					END_IF

				END_IF

			PATLITE_STATE_ERROR:

				IF ErrorCount > ERROR_COUNT_THRESH THEN
					CommError := TRUE;
				END_IF

				CommState := PATLITE_STATE_WRITE_REGISTER;

		END_CASE

		IF(EDGEPOS(CommError)) THEN
			MpAlarmXSet(gAlarmXCore, ALARM_PATLITE_COMMS);
		ELSIF (EDGENEG(CommError)) THEN
			MpAlarmXReset(gAlarmXCore, ALARM_PATLITE_COMMS);
		END_IF
	END_IF

END_PROGRAM
```

#### Patelite.typ - Local data types
```iecst
(********************************************************************
 * COPYRIGHT -- Bernecker + Rainer
 ********************************************************************
 * Program: MbApp
 * File: MbApp.typ
 * Author: Bernecker + Rainer
 * Created: October 22, 2009
 ********************************************************************
 * Local data types of program MbApp
 ********************************************************************)

TYPE
	CommStateEnum :
		(
		PATLITE_STATE_STANDBY,
		PATLITE_STATE_WRITE_REGISTER,
		PATLITE_STATE_ERROR
		);
	GroupEnum :
		(
		GROUP_1_POWER_ON,
		GROUP_2_HEATING,
		GROUP_3_HEAT_AIR_OK,
		GROUP_4_RUN,
		GROUP_5_SAFETY
		);
END_TYPE
```

#### Patelite.var - Local variables
```iecst
(********************************************************************
 * COPYRIGHT -- Bernecker + Rainer
 ********************************************************************
 * Program: MbApp
 * File: MbApp.var
 * Author: Bernecker + Rainer
 * Created: October 22, 2009
 ********************************************************************
 * Local variables of program MbApp
 ********************************************************************)
VAR CONSTANT
	GROUP_OFFSET : UINT := 257;
END_VAR
VAR
	CommState : CommStateEnum;
	NextLightGroup : GroupEnum;
	CurrentLightGroup : GroupEnum;
	mbWriteSingleRegister_0 : mbWriteSingleRegister; (*function block structure*)
END_VAR
VAR CONSTANT
	GROUP_REG_ADR : UINT := 6; (*register address for light group on modbus station*)
END_VAR
VAR
	mb_station : STRING[20]; (*path to modbus station*)
	ErrorCount : UINT;
END_VAR
VAR CONSTANT
	ERROR_COUNT_THRESH : UINT := 10;
END_VAR
VAR
	CommError : BOOL;
END_VAR
```

### Package Logical/AsSafetySolution - AsSafety design sample

- Button.clm (not shown)

- button.fninfo (not shown)

- Default.fninfo (not shown)

- header.fninfo (not shown)

- Html_SDM.fninfo (not shown)

- info.fninfo (not shown)

- Input.fninfo (not shown)

- status.fninfo (not shown)

- Background.layer (not shown)

- globalArea.layer (not shown)

- msgBox.layer (not shown)

- Trend_Temperature.tre (not shown)

### Program Logical/AsSafetySolution/SafetySample

#### SafetySample.var
```iecst
(********************************************************************
 * COPYRIGHT -- Bernecker + Rainer
 ********************************************************************
 * Program: SafetySample
 * File: SafetySample.var
 * Author: B&R
 ********************************************************************
 * Local variables of program SafetySample
 ********************************************************************)
VAR
	appcmd1 : DownloadCmdApplicationTypeV1; (*command structure for application download*)
	dataAcknMachineOptions : DownloadAcknMaOpTypeV1; (*data to acknowledge bit machine options*)
	datacmd1 : DownloadCmdMaOpTypeV1; (*command structure for machine options download*)
	datacmd2 : DownloadCmdExtMaOpTypeV1; (*command structure for extended machine options download*)
	dataMachineOptionsBitInput : ConfigurationBitOptionsTypeV1; (*data for bit machine options*)
	dataModuleFlagsInput : ConfigurationModuleFlagsTypeV1; (*data for module flags*)
	dialogApplication : BOOL; (*visualization dialog for application download*)
	dialogButtonLeft : BOOL; (*left button in visualization dialog*)
	dialogButtonRight : BOOL; (*right button in visualization dialog*)
	dialogData : BOOL; (*visualization dialog for machine options download*)
	dialogExtData : BOOL; (*visualization dialog for extended machine options download*)
	dialogRemoteCmd : BOOL; (*visualization dialog for remote control*)
	executeapp1 : BOOL; (*execute application download*)
	executedata1 : BOOL; (*execute machine options download*)
	executedata2 : BOOL; (*execute extended machine options download*)
	executeRemoteCmd : BOOL; (*execute remote control*)
	indexButtonLeft : UINT; (*index for button text*)
	indexButtonRight : UINT; (* index for button text*)
	indexCompareTextData : UINT; (*index for compare message machine options*)
	indexCompareTextExtData : UINT; (*index for compare message extended machine options*)
	indexFAILLed : UINT; (*index FAIL led*)
	indexFwAcknLed : UINT; (*index FW-ACKN led*)
	indexHeaderText : UINT; (*index dialog header text*)
	indexMessageText : UINT; (*index message text*)
	indexMxchgLed : UINT; (*index MXCHG led*)
	indexRELed : UINT; (*index R/E led*)
	Interface : STRING[80] := 'IF3'; (*interface information for SafeLOGIC*)
	Node : USINT := 1; (*node information for SafeLOGIC*)
	pDeviceListOut : REFERENCE TO ARRAY[0..1] OF ConfigurationDeviceTypeV1; (*device list from FUB*)
	pMachineOptionsBitOut : REFERENCE TO ConfigurationBitOptionsTypeV1; (*bit machine options from FUB*)
	pModuleFlagsOut : REFERENCE TO ConfigurationModuleFlagsTypeV1; (*module flags form FUB*)
	readUDIDhighSL : EplSDORead; (*function block to read UDID high from device*)
	readUDIDhighSLX : AsIOAccRead; (*function block to read UDID high from device*)
	readUDIDlowSL : EplSDORead; (*function block to read UDID low from device*)
	readUDIDlowSLX : AsIOAccRead; (*function block to read UDID low from device*)
	remotecmd : RemoteControlCmdTypeV1; (*command structure for remote control*)
	safeDownloadApplication_0 : safeDownloadApplication; (*function block safeDownloadApplication*)
	safeDownloadData_0 : safeDownloadData; (*function block safeDownloadData*)
	safeDownloadData_1 : safeDownloadData; (*function block safeDownloadData*)
	safeRemoteControl_0 : safeRemoteControl; (*function block safeRemoteControl*)
	slxused : BOOL; (*SafeLOGIC-X is used*)
	Station : STRING[80] := 'IF6.ST3'; (*station information for SafeLOGIC-X*)
	statusAcknInfoData : UINT; (*acknowledge boxes for machine options*)
	statusAcknInfoExtData : UINT; (*acknowledge boxes for extended machine options*)
	statusButtonActiv : ARRAY[0..15] OF USINT; (*button activ*)
	statusButtonInactiv : ARRAY[0..15] OF USINT; (*button inactiv*)
	statusButtonUnlockApp : UINT; (*unlock buttons application*)
	statusButtonUnlockData : UINT; (*unlock buttons data*)
	statusButtonUnlockExtData : UINT; (*unlock buttons extended data*)
	statusDialog : UINT; (*dialog box*)
	statusSetPassword : UINT; (*visualization status to set password*)
	statusSLInformation : UINT; (*display information for SafeLOGIC*)
	stautsSLXInformation : UINT; (*display information for SafeLOGIC-X*)
	UDID_High : UINT; (*UDID_high for SafelOGIC*)
	UDID_Low : UDINT; (*UDID_low for SafeLOGIC*)
	visuAcknExtData : DownloadAcknExtMaOpTypeV1; (*acknowledge extended machine options*)
	visuAcknMachineOptions : ARRAY[0..511] OF BOOL; (*acknowledge machine options*)
	visuApplicationCRC : STRING[8]; (*CRC HEX string for visualization*)
	visuDeviceListInput : ARRAY[0..1] OF DownloadDeviceTypeV1; (*device list input*)
	visuDeviceListOutput : ARRAY[0..1] OF DownloadDeviceTypeV1; (*device list output*)
	visuDintInput : ConfigurationDintOptionsTypeV1; (*DINT channels input*)
	visuDintOutput : ConfigurationDintOptionsTypeV1; (*DINT channels output*)
	visuEnableDINTOptions : BOOL; (*enable DINT options*)
	visuEnableINTOptions : BOOL; (*enable INT options*)
	visuEnableMachineOptions : BOOL; (*enable BIT options*)
	visuEnableModuleFlags : BOOL; (*enable module flags*)
	visuEnableUDINTOptions : BOOL; (*enable UDINT options*)
	visuEnableUINTOptions : BOOL; (*enable UINT options*)
	visuIntInput : ConfigurationIntOptionsTypeV1; (*INT channels input*)
	visuIntOutput : ConfigurationIntOptionsTypeV1; (*INT channels output*)
	visuMachineOptionsBitInput : ARRAY[0..511] OF BOOL; (*BIT options input*)
	visuMachineOptionsBitOutput : ARRAY[0..511] OF BOOL; (*BIT options output*)
	visuModuleFlagsNotPresentInput : ARRAY[0..1023] OF BOOL; (*not present module flags input*)
	visuModuleFlagsNotPresentOutput : ARRAY[0..1023] OF BOOL; (*not present module flags output*)
	visuModuleFlagsOptionalInput : ARRAY[0..1023] OF BOOL; (*optional module flags input*)
	visuModuleFlagsOptionalOutput : ARRAY[0..1023] OF BOOL; (*optional module flags output*)
	visuModuleFlagsStartupInput : ARRAY[0..1023] OF BOOL; (*startup module flags input*)
	visuModuleFlagsStartupOutput : ARRAY[0..1023] OF BOOL; (*startup module flags output*)
	visuUDID_High : STRING[8]; (*UDID hex string for visualization*)
	visuUDID_Low : STRING[8]; (*UDID hex string for visualization*)
	visuUdintInput : ConfigurationUdintOptionsTypeV1; (*UDINT channels input*)
	visuUdintOutput : ConfigurationUdintOptionsTypeV1; (*UDINT channels output*)
	visuUintInput : ConfigurationUintOptionsTypeV1; (*UINT channels input*)
	visuUintOutput : ConfigurationUintOptionsTypeV1; (*UINT channels output*)
	visuUsedSLIDData : UINT; (*SafeLOGIC ID for data download*)
	visuUsedSLIDRemote : UINT; (*SafeLOGIC ID for remote control*)
	xcnt : UINT; (*counter variable*)
	visuLockSDP : INT;
END_VAR
```
